LIN {X 0,Y 350.483,Z 210.53,A -85,B 0,C 180,E1 -14687.75,E2 -14687.75} C_VEL
LIN {X 0,Y 348.097,Z 207.912,A -85,B 0,C 180,E1 -14688.285,E2 -14688.285} C_VEL
LIN {X 0,Y 344.862,Z 203.942,A -85,B 0,C 180,E1 -14688.984,E2 -14688.984} C_VEL
LIN {X 0,Y 341.244,Z 199.767,A -85,B 0,C 180,E1 -14689.717,E2 -14689.717} C_VEL
LIN {X 0,Y 339.454,Z 197.486,A -85,B 0,C 180,E1 -14690.077,E2 -14690.077} C_VEL
LIN {X 0,Y 337.301,Z 194.627,A -85,B 0,C 180,E1 -14690.498,E2 -14690.498} C_VEL
LIN {X 0,Y 336.134,Z 192.909,A -85,B 0,C 180,E1 -14690.724,E2 -14690.724} C_VEL
LIN {X 0,Y 334.391,Z 190.698,A -85,B 0,C 180,E1 -14691.054,E2 -14691.054} C_VEL
LIN {X 0,Y 333.682,Z 188.419,A -85,B 0,C 180,E1 -14691.257,E2 -14691.257} C_VEL
LIN {X 0,Y 333.715,Z 188.414,A -85,B 0,C 180,E1 -14695.101,E2 -14695.101} C_VEL
LIN {X 0,Y 333.718,Z 188.416,A -85,B 0,C 180,E1 -14697.811,E2 -14697.811} C_VEL
LIN {X 0,Y 333.695,Z 188.419,A -85,B 0,C 180,E1 -14700.362,E2 -14700.362} C_VEL
LIN {X 0,Y 333.669,Z 188.42,A -85,B 0,C 180,E1 -14704.659,E2 -14704.659} C_VEL
LIN {X 0,Y 333.652,Z 188.425,A -85,B 0,C 180,E1 -14707.65,E2 -14707.65} C_VEL
LIN {X 0,Y 333.65,Z 188.421,A -85,B 0,C 180,E1 -14710.766,E2 -14710.766} C_VEL
LIN {X 0,Y 333.598,Z 188.429,A -85,B 0,C 180,E1 -14714.252,E2 -14714.252} C_VEL
LIN {X 0,Y 333.663,Z 188.425,A -85,B 0,C 180,E1 -14717.623,E2 -14717.623} C_VEL
LIN {X 0,Y 333.672,Z 188.422,A -85,B 0,C 180,E1 -14721.197,E2 -14721.197} C_VEL
LIN {X 0,Y 333.68,Z 188.422,A -85,B 0,C 180,E1 -14725.226,E2 -14725.226} C_VEL
LIN {X 0,Y 333.692,Z 188.418,A -85,B 0,C 180,E1 -14729.638,E2 -14729.638} C_VEL
LIN {X 0,Y 333.739,Z 188.411,A -85,B 0,C 180,E1 -14732.402,E2 -14732.402} C_VEL
LIN {X 0,Y 333.721,Z 188.417,A -85,B 0,C 180,E1 -14735.091,E2 -14735.091} C_VEL
LIN {X 0,Y 333.68,Z 188.421,A -85,B 0,C 180,E1 -14739.02,E2 -14739.02} C_VEL
LIN {X 0,Y 333.699,Z 188.414,A -85,B 0,C 180,E1 -14739.925,E2 -14739.925} C_VEL
LIN {X 0,Y 333.087,Z 188.496,A -85,B 0,C 180,E1 -14740.932,E2 -14740.932} C_VEL
LIN {X 0,Y 330.262,Z 188.848,A -85,B 0,C 180,E1 -14742.571,E2 -14742.571} C_VEL
LIN {X 0,Y 327.848,Z 189.149,A -85,B 0,C 180,E1 -14743.899,E2 -14743.899} C_VEL
LIN {X 0,Y 326.826,Z 189.275,A -85,B 0,C 180,E1 -14744.927,E2 -14744.927} C_VEL
LIN {X 0,Y 326.752,Z 189.281,A -85,B 0,C 180,E1 -14745.275,E2 -14745.275} C_VEL
LIN {X 0,Y 326.764,Z 189.282,A -85,B 0,C 180,E1 -14748.839,E2 -14748.839} C_VEL
LIN {X 0,Y 326.953,Z 189.261,A -85,B 0,C 180,E1 -14752.59,E2 -14752.59} C_VEL
LIN {X 0,Y 326.77,Z 189.277,A -85,B 0,C 180,E1 -14755.065,E2 -14755.065} C_VEL
LIN {X 0,Y 327.041,Z 189.24,A -85,B 0,C 180,E1 -14757.537,E2 -14757.537} C_VEL
LIN {X 0,Y 327.193,Z 189.225,A -85,B 0,C 180,E1 -14760.001,E2 -14760.001} C_VEL
LIN {X 0,Y 327.04,Z 189.248,A -85,B 0,C 180,E1 -14762.464,E2 -14762.464} C_VEL
LIN {X 0,Y 326.984,Z 189.257,A -85,B 0,C 180,E1 -14766.17,E2 -14766.17} C_VEL
LIN {X 0,Y 326.802,Z 189.279,A -85,B 0,C 180,E1 -14769.907,E2 -14769.907} C_VEL
LIN {X 0,Y 326.755,Z 189.284,A -85,B 0,C 180,E1 -14773.686,E2 -14773.686} C_VEL
LIN {X 0,Y 326.696,Z 189.291,A -85,B 0,C 180,E1 -14777.529,E2 -14777.529} C_VEL
LIN {X 0,Y 326.659,Z 189.294,A -85,B 0,C 180,E1 -14780.136,E2 -14780.136} C_VEL
LIN {X 0,Y 326.65,Z 189.295,A -85,B 0,C 180,E1 -14784.13,E2 -14784.13} C_VEL
LIN {X 0,Y 326.68,Z 189.291,A -85,B 0,C 180,E1 -14786.859,E2 -14786.859} C_VEL
LIN {X 0,Y 326.632,Z 189.297,A -85,B 0,C 180,E1 -14790.61,E2 -14790.61} C_VEL
LIN {X 0,Y 326.605,Z 189.302,A -85,B 0,C 180,E1 -14794.02,E2 -14794.02} C_VEL
LIN {X 0,Y 326.685,Z 189.697,A -85,B 0,C 180,E1 -14795.511,E2 -14795.511} C_VEL
LIN {X 0,Y 327.059,Z 192.418,A -85,B 0,C 180,E1 -14799.324,E2 -14799.324} C_VEL
LIN {X 0,Y 327.355,Z 194.259,A -85,B 0,C 180,E1 -14801.725,E2 -14801.725} C_VEL
LIN {X 0,Y 327.712,Z 196.982,A -85,B 0,C 180,E1 -14805.049,E2 -14805.049} C_VEL
LIN {X 0,Y 327.836,Z 199.974,A -85,B 0,C 180,E1 -14808.352,E2 -14808.352} C_VEL
LIN {X 0,Y 327.498,Z 203.094,A -85,B 0,C 180,E1 -14811.514,E2 -14811.514} C_VEL
LIN {X 0,Y 327.023,Z 206.495,A -85,B 0,C 180,E1 -14814.752,E2 -14814.752} C_VEL
LIN {X 0,Y 326.604,Z 209.457,A -85,B 0,C 180,E1 -14817.456,E2 -14817.456} C_VEL
LIN {X 0,Y 326.202,Z 212.67,A -85,B 0,C 180,E1 -14820.296,E2 -14820.296} C_VEL
LIN {X 0,Y 325.859,Z 215.915,A -85,B 0,C 180,E1 -14823.069,E2 -14823.069} C_VEL
LIN {X 0,Y 325.459,Z 220.798,A -85,B 0,C 180,E1 -14827.127,E2 -14827.127} C_VEL
LIN {X 0,Y 325.414,Z 221.412,A -85,B 0,C 180,E1 -14827.655,E2 -14827.655} C_VEL
LIN {X 0,Y 327.617,Z 230.715,A -85,B 0,C 180,E1 -14828.173,E2 -14828.173} C_VEL
LIN {X 0,Y 329.57,Z 240.233,A -85,B 0,C 180,E1 -14828.813,E2 -14828.813} C_VEL
LIN {X 0,Y 331.05,Z 249.851,A -85,B 0,C 180,E1 -14829.573,E2 -14829.573} C_VEL
LIN {X 0,Y 332.04,Z 258.46,A -85,B 0,C 180,E1 -14830.366,E2 -14830.366} C_VEL
LIN {X 0,Y 332.381,Z 263.384,A -85,B 0,C 180,E1 -14830.869,E2 -14830.869} C_VEL
LIN {X 0,Y 330.862,Z 275.575,A -85,B 0,C 180,E1 -14832.221,E2 -14832.221} C_VEL
LIN {X 0,Y 329.888,Z 283.327,A -85,B 0,C 180,E1 -14833.286,E2 -14833.286} C_VEL
LIN {X 0,Y 328.677,Z 292.466,A -85,B 0,C 180,E1 -14834.815,E2 -14834.815} C_VEL
LIN {X 0,Y 327.865,Z 298.672,A -85,B 0,C 180,E1 -14836.046,E2 -14836.046} C_VEL
LIN {X 0,Y 326.878,Z 305.21,A -85,B 0,C 180,E1 -14837.584,E2 -14837.584} C_VEL
LIN {X 0,Y 326.347,Z 309.716,A -85,B 0,C 180,E1 -14838.824,E2 -14838.824} C_VEL
LIN {X 0,Y 325.644,Z 315.21,A -85,B 0,C 180,E1 -14840.685,E2 -14840.685} C_VEL
LIN {X 0,Y 325.21,Z 319.539,A -85,B 0,C 180,E1 -14842.55,E2 -14842.55} C_VEL
LIN {X 0,Y 324.998,Z 322.39,A -85,B 0,C 180,E1 -14844.125,E2 -14844.125} C_VEL
LIN {X 0,Y 324.912,Z 325.1,A -85,B 0,C 180,E1 -14846.279,E2 -14846.279} C_VEL
LIN {X 0,Y 324.838,Z 326.158,A -85,B 0,C 180,E1 -14847.52,E2 -14847.52} C_VEL
LIN {X 0,Y 324.815,Z 326.747,A -85,B 0,C 180,E1 -14848.76,E2 -14848.76} C_VEL
LIN {X 0,Y 324.815,Z 326.747,A -85,B 0,C 180,E1 -14851.24,E2 -14851.24} C_VEL
LIN {X 0,Y 324.838,Z 326.158,A -85,B 0,C 180,E1 -14852.48,E2 -14852.48} C_VEL
LIN {X 0,Y 324.931,Z 323.709,A -85,B 0,C 180,E1 -14854.963,E2 -14854.963} C_VEL
LIN {X 0,Y 325.121,Z 320.757,A -85,B 0,C 180,E1 -14856.828,E2 -14856.828} C_VEL
LIN {X 0,Y 325.474,Z 316.766,A -85,B 0,C 180,E1 -14858.694,E2 -14858.694} C_VEL
LIN {X 0,Y 326.08,Z 311.633,A -85,B 0,C 180,E1 -14860.556,E2 -14860.556} C_VEL
LIN {X 0,Y 326.724,Z 306.367,A -85,B 0,C 180,E1 -14862.106,E2 -14862.106} C_VEL
LIN {X 0,Y 327.646,Z 300.048,A -85,B 0,C 180,E1 -14863.647,E2 -14863.647} C_VEL
LIN {X 0,Y 328.437,Z 294.094,A -85,B 0,C 180,E1 -14864.879,E2 -14864.879} C_VEL
LIN {X 0,Y 329.422,Z 287.165,A -85,B 0,C 180,E1 -14866.102,E2 -14866.102} C_VEL
LIN {X 0,Y 330.396,Z 278.98,A -85,B 0,C 180,E1 -14867.325,E2 -14867.325} C_VEL
LIN {X 0,Y 331.502,Z 270.468,A -85,B 0,C 180,E1 -14868.382,E2 -14868.382} C_VEL
LIN {X 0,Y 332.359,Z 263.383,A -85,B 0,C 180,E1 -14869.133,E2 -14869.133} C_VEL
LIN {X 0,Y 331.643,Z 254.402,A -85,B 0,C 180,E1 -14870.026,E2 -14870.026} C_VEL
LIN {X 0,Y 330.252,Z 244.324,A -85,B 0,C 180,E1 -14870.884,E2 -14870.884} C_VEL
LIN {X 0,Y 328.126,Z 233.062,A -85,B 0,C 180,E1 -14871.682,E2 -14871.682} C_VEL
LIN {X 0,Y 325.67,Z 223.147,A -85,B 0,C 180,E1 -14872.27,E2 -14872.27} C_VEL
LIN {X 0,Y 325.411,Z 221.414,A -85,B 0,C 180,E1 -14872.344,E2 -14872.344} C_VEL
LIN {X 0,Y 325.716,Z 217.555,A -85,B 0,C 180,E1 -14875.565,E2 -14875.565} C_VEL
LIN {X 0,Y 326.057,Z 214.284,A -85,B 0,C 180,E1 -14878.307,E2 -14878.307} C_VEL
LIN {X 0,Y 326.604,Z 209.433,A -85,B 0,C 180,E1 -14882.544,E2 -14882.544} C_VEL
LIN {X 0,Y 327.05,Z 206.248,A -85,B 0,C 180,E1 -14885.464,E2 -14885.464} C_VEL
LIN {X 0,Y 327.497,Z 203.094,A -85,B 0,C 180,E1 -14888.486,E2 -14888.486} C_VEL
LIN {X 0,Y 327.829,Z 199.972,A -85,B 0,C 180,E1 -14891.649,E2 -14891.649} C_VEL
LIN {X 0,Y 327.833,Z 198.426,A -85,B 0,C 180,E1 -14893.314,E2 -14893.314} C_VEL
LIN {X 0,Y 327.512,Z 195.562,A -85,B 0,C 180,E1 -14896.631,E2 -14896.631} C_VEL
LIN {X 0,Y 327.137,Z 193.006,A -85,B 0,C 180,E1 -14899.871,E2 -14899.871} C_VEL
LIN {X 0,Y 326.805,Z 190.726,A -85,B 0,C 180,E1 -14902.976,E2 -14902.976} C_VEL
LIN {X 0,Y 326.67,Z 189.471,A -85,B 0,C 180,E1 -14904.837,E2 -14904.837} C_VEL
LIN {X 0,Y 326.606,Z 189.302,A -85,B 0,C 180,E1 -14907.455,E2 -14907.455} C_VEL
LIN {X 0,Y 326.646,Z 189.298,A -85,B 0,C 180,E1 -14910.339,E2 -14910.339} C_VEL
LIN {X 0,Y 326.688,Z 189.295,A -85,B 0,C 180,E1 -14914.515,E2 -14914.515} C_VEL
LIN {X 0,Y 326.643,Z 189.299,A -85,B 0,C 180,E1 -14918.544,E2 -14918.544} C_VEL
LIN {X 0,Y 326.742,Z 189.282,A -85,B 0,C 180,E1 -14921.177,E2 -14921.177} C_VEL
LIN {X 0,Y 326.76,Z 189.28,A -85,B 0,C 180,E1 -14925.432,E2 -14925.432} C_VEL
LIN {X 0,Y 326.766,Z 189.279,A -85,B 0,C 180,E1 -14928.838,E2 -14928.838} C_VEL
LIN {X 0,Y 326.953,Z 189.256,A -85,B 0,C 180,E1 -14932.589,E2 -14932.589} C_VEL
LIN {X 0,Y 326.769,Z 189.279,A -85,B 0,C 180,E1 -14935.064,E2 -14935.064} C_VEL
LIN {X 0,Y 327.04,Z 189.248,A -85,B 0,C 180,E1 -14937.536,E2 -14937.536} C_VEL
LIN {X 0,Y 327.193,Z 189.225,A -85,B 0,C 180,E1 -14939.999,E2 -14939.999} C_VEL
LIN {X 0,Y 327.041,Z 189.24,A -85,B 0,C 180,E1 -14942.463,E2 -14942.463} C_VEL
LIN {X 0,Y 326.954,Z 189.255,A -85,B 0,C 180,E1 -14946.646,E2 -14946.646} C_VEL
LIN {X 0,Y 326.8,Z 189.275,A -85,B 0,C 180,E1 -14949.906,E2 -14949.906} C_VEL
LIN {X 0,Y 326.754,Z 189.281,A -85,B 0,C 180,E1 -14953.685,E2 -14953.685} C_VEL
LIN {X 0,Y 326.694,Z 189.29,A -85,B 0,C 180,E1 -14957.527,E2 -14957.527} C_VEL
LIN {X 0,Y 326.66,Z 189.29,A -85,B 0,C 180,E1 -14960.134,E2 -14960.134} C_VEL
LIN {X 0,Y 326.646,Z 189.293,A -85,B 0,C 180,E1 -14964.128,E2 -14964.128} C_VEL
LIN {X 0,Y 326.68,Z 189.294,A -85,B 0,C 180,E1 -14966.857,E2 -14966.857} C_VEL
LIN {X 0,Y 326.633,Z 189.299,A -85,B 0,C 180,E1 -14970.611,E2 -14970.611} C_VEL
LIN {X 0,Y 326.601,Z 189.3,A -85,B 0,C 180,E1 -14974.019,E2 -14974.019} C_VEL
LIN {X 0,Y 326.624,Z 189.297,A -85,B 0,C 180,E1 -14977.239,E2 -14977.239} C_VEL
LIN {X 0,Y 326.598,Z 189.303,A -85,B 0,C 180,E1 -14980.207,E2 -14980.207} C_VEL
LIN {X 0,Y 326.566,Z 189.304,A -85,B 0,C 180,E1 -14983.524,E2 -14983.524} C_VEL
LIN {X 0,Y 326.571,Z 189.303,A -85,B 0,C 180,E1 -14987.028,E2 -14987.028} C_VEL
LIN {X 0,Y 326.606,Z 189.3,A -85,B 0,C 180,E1 -14990.773,E2 -14990.773} C_VEL
LIN {X 0,Y 326.608,Z 189.301,A -85,B 0,C 180,E1 -14994.48,E2 -14994.48} C_VEL
LIN {X 0,Y 326.61,Z 189.3,A -85,B 0,C 180,E1 -14997.456,E2 -14997.456} C_VEL
LIN {X 0,Y 326.657,Z 189.295,A -85,B 0,C 180,E1 -15000.341,E2 -15000.341} C_VEL
LIN {X 0,Y 326.681,Z 189.291,A -85,B 0,C 180,E1 -15003.143,E2 -15003.143} C_VEL
LIN {X 0,Y 326.648,Z 189.299,A -85,B 0,C 180,E1 -15005.871,E2 -15005.871} C_VEL
LIN {X 0,Y 326.654,Z 189.298,A -85,B 0,C 180,E1 -15007.82,E2 -15007.82} C_VEL
LIN {X 0,Y 327.795,Z 192.347,A -85,B 0,C 180,E1 -15008.061,E2 -15008.061} C_VEL
LIN {X 0,Y 329.517,Z 194.65,A -85,B 0,C 180,E1 -15008.362,E2 -15008.362} C_VEL
LIN {X 0,Y 331.953,Z 198.098,A -85,B 0,C 180,E1 -15008.797,E2 -15008.797} C_VEL
LIN {X 0,Y 335.943,Z 203.215,A -85,B 0,C 180,E1 -15009.532,E2 -15009.532} C_VEL
LIN {X 0,Y 340.414,Z 208.614,A -85,B 0,C 180,E1 -15010.402,E2 -15010.402} C_VEL
LIN {X 0,Y 345.28,Z 214.213,A -85,B 0,C 180,E1 -15011.406,E2 -15011.406} C_VEL
LIN {X 0,Y 347.897,Z 217.095,A -85,B 0,C 180,E1 -15011.984,E2 -15011.984} C_VEL
LIN {X 0,Y 352.051,Z 221.223,A -85,B 0,C 180,E1 -15012.932,E2 -15012.932} C_VEL
LIN {X 0,Y 356.881,Z 226.359,A -85,B 0,C 180,E1 -15014.144,E2 -15014.144} C_VEL
LIN {X 0,Y 360.132,Z 229.27,A -85,B 0,C 180,E1 -15015.015,E2 -15015.015} C_VEL
LIN {X 0,Y 364.662,Z 233.73,A -85,B 0,C 180,E1 -15016.357,E2 -15016.357} C_VEL
LIN {X 0,Y 367.666,Z 236.169,A -85,B 0,C 180,E1 -15017.32,E2 -15017.32} C_VEL
LIN {X 0,Y 370.754,Z 239.393,A -85,B 0,C 180,E1 -15018.471,E2 -15018.471} C_VEL
LIN {X 0,Y 372.501,Z 240.811,A -85,B 0,C 180,E1 -15019.125,E2 -15019.125} C_VEL
LIN {X 0,Y 375.48,Z 242.667,A -85,B 0,C 180,E1 -15020.302,E2 -15020.302} C_VEL
LIN {X 0,Y 377.708,Z 245.024,A -85,B 0,C 180,E1 -15021.44,E2 -15021.44} C_VEL
LIN {X 0,Y 379.626,Z 247.006,A -85,B 0,C 180,E1 -15022.554,E2 -15022.554} C_VEL
LIN {X 0,Y 381.687,Z 248.584,A -85,B 0,C 180,E1 -15023.874,E2 -15023.874} C_VEL
LIN {X 0,Y 382.853,Z 249.33,A -85,B 0,C 180,E1 -15024.734,E2 -15024.734} C_VEL
LIN {X 0,Y 384.103,Z 249.928,A -85,B 0,C 180,E1 -15025.803,E2 -15025.803} C_VEL
LIN {X 0,Y 385.142,Z 250.169,A -85,B 0,C 180,E1 -15026.862,E2 -15026.862} C_VEL
LIN {X 0,Y 385.884,Z 250.348,A -85,B 0,C 180,E1 -15027.913,E2 -15027.913} C_VEL
LIN {X 0,Y 386.362,Z 250.4,A -85,B 0,C 180,E1 -15028.958,E2 -15028.958} C_VEL
LIN {X 0,Y 386.509,Z 250.455,A -85,B 0,C 180,E1 -15030,E2 -15030} C_VEL
LIN {X 0,Y 386.362,Z 250.371,A -85,B 0,C 180,E1 -15031.042,E2 -15031.042} C_VEL
LIN {X 0,Y 385.884,Z 250.332,A -85,B 0,C 180,E1 -15032.087,E2 -15032.087} C_VEL
LIN {X 0,Y 385.152,Z 250.141,A -85,B 0,C 180,E1 -15033.138,E2 -15033.138} C_VEL
LIN {X 0,Y 384.128,Z 249.9,A -85,B 0,C 180,E1 -15034.197,E2 -15034.197} C_VEL
LIN {X 0,Y 382.819,Z 249.345,A -85,B 0,C 180,E1 -15035.267,E2 -15035.267} C_VEL
LIN {X 0,Y 381.358,Z 248.36,A -85,B 0,C 180,E1 -15036.348,E2 -15036.348} C_VEL
LIN {X 0,Y 379.625,Z 246.957,A -85,B 0,C 180,E1 -15037.446,E2 -15037.446} C_VEL
LIN {X 0,Y 377.041,Z 244.248,A -85,B 0,C 180,E1 -15038.922,E2 -15038.922} C_VEL
LIN {X 0,Y 375.403,Z 242.649,A -85,B 0,C 180,E1 -15039.7,E2 -15039.7} C_VEL
LIN {X 0,Y 372.239,Z 240.59,A -85,B 0,C 180,E1 -15040.959,E2 -15040.959} C_VEL
LIN {X 0,Y 368.635,Z 237.327,A -85,B 0,C 180,E1 -15042.312,E2 -15042.312} C_VEL
LIN {X 0,Y 366.406,Z 235.019,A -85,B 0,C 180,E1 -15043.098,E2 -15043.098} C_VEL
LIN {X 0,Y 362.568,Z 231.873,A -85,B 0,C 180,E1 -15044.261,E2 -15044.261} C_VEL
LIN {X 0,Y 358.361,Z 227.539,A -85,B 0,C 180,E1 -15045.468,E2 -15045.468} C_VEL
LIN {X 0,Y 354.273,Z 223.764,A -85,B 0,C 180,E1 -15046.513,E2 -15046.513} C_VEL
LIN {X 0,Y 351.124,Z 220.432,A -85,B 0,C 180,E1 -15047.28,E2 -15047.28} C_VEL
LIN {X 0,Y 346.949,Z 215.921,A -85,B 0,C 180,E1 -15048.238,E2 -15048.238} C_VEL
LIN {X 0,Y 342.082,Z 210.601,A -85,B 0,C 180,E1 -15049.26,E2 -15049.26} C_VEL
LIN {X 0,Y 339.011,Z 207.141,A -85,B 0,C 180,E1 -15049.871,E2 -15049.871} C_VEL
LIN {X 0,Y 335.427,Z 202.682,A -85,B 0,C 180,E1 -15050.562,E2 -15050.562} C_VEL
LIN {X 0,Y 332.765,Z 198.959,A -85,B 0,C 180,E1 -15051.067,E2 -15051.067} C_VEL
LIN {X 0,Y 329.9,Z 195.384,A -85,B 0,C 180,E1 -15051.562,E2 -15051.562} C_VEL
LIN {X 0,Y 328.729,Z 193.458,A -85,B 0,C 180,E1 -15051.78,E2 -15051.78} C_VEL
LIN {X 0,Y 327.241,Z 191.338,A -85,B 0,C 180,E1 -15052.037,E2 -15052.037} C_VEL
LIN {X 0,Y 326.661,Z 189.297,A -85,B 0,C 180,E1 -15052.205,E2 -15052.205} C_VEL
LIN {X 0,Y 326.686,Z 189.29,A -85,B 0,C 180,E1 -15055.484,E2 -15055.484} C_VEL
LIN {X 0,Y 326.668,Z 189.296,A -85,B 0,C 180,E1 -15058.249,E2 -15058.249} C_VEL
LIN {X 0,Y 326.596,Z 189.3,A -85,B 0,C 180,E1 -15061.094,E2 -15061.094} C_VEL
LIN {X 0,Y 326.604,Z 189.304,A -85,B 0,C 180,E1 -15064.019,E2 -15064.019} C_VEL
LIN {X 0,Y 326.626,Z 189.297,A -85,B 0,C 180,E1 -15067.239,E2 -15067.239} C_VEL
LIN {X 0,Y 326.599,Z 189.302,A -85,B 0,C 180,E1 -15070.207,E2 -15070.207} C_VEL
LIN {X 0,Y 326.573,Z 189.306,A -85,B 0,C 180,E1 -15073.523,E2 -15073.523} C_VEL
LIN {X 0,Y 326.589,Z 189.302,A -85,B 0,C 180,E1 -15077.025,E2 -15077.025} C_VEL
LIN {X 0,Y 326.629,Z 189.296,A -85,B 0,C 180,E1 -15080.768,E2 -15080.768} C_VEL
LIN {X 0,Y 326.607,Z 189.299,A -85,B 0,C 180,E1 -15084.481,E2 -15084.481} C_VEL
LIN {X 0,Y 326.602,Z 189.303,A -85,B 0,C 180,E1 -15087.456,E2 -15087.456} C_VEL
LIN {X 0,Y 326.655,Z 189.293,A -85,B 0,C 180,E1 -15090.341,E2 -15090.341} C_VEL
LIN {X 0,Y 326.685,Z 189.289,A -85,B 0,C 180,E1 -15094.517,E2 -15094.517} C_VEL
LIN {X 0,Y 326.643,Z 189.296,A -85,B 0,C 180,E1 -15098.546,E2 -15098.546} C_VEL
LIN {X 0,Y 326.739,Z 189.285,A -85,B 0,C 180,E1 -15101.178,E2 -15101.178} C_VEL
LIN {X 0,Y 326.752,Z 189.281,A -85,B 0,C 180,E1 -15105.275,E2 -15105.275} C_VEL
LIN {X 0,Y 326.102,Z 189.364,A -85,B 0,C 180,E1 -15106.304,E2 -15106.304} C_VEL
LIN {X 0,Y 323.235,Z 189.719,A -85,B 0,C 180,E1 -15107.978,E2 -15107.978} C_VEL
LIN {X 0,Y 320.826,Z 190.018,A -85,B 0,C 180,E1 -15109.335,E2 -15109.335} C_VEL
LIN {X 0,Y 319.841,Z 190.144,A -85,B 0,C 180,E1 -15110.386,E2 -15110.386} C_VEL
LIN {X 0,Y 319.788,Z 190.146,A -85,B 0,C 180,E1 -15110.741,E2 -15110.741} C_VEL
LIN {X 0,Y 319.939,Z 190.129,A -85,B 0,C 180,E1 -15113.695,E2 -15113.695} C_VEL
LIN {X 0,Y 319.985,Z 190.117,A -85,B 0,C 180,E1 -15117.483,E2 -15117.483} C_VEL
LIN {X 0,Y 320.145,Z 190.102,A -85,B 0,C 180,E1 -15120.001,E2 -15120.001} C_VEL
LIN {X 0,Y 319.984,Z 190.127,A -85,B 0,C 180,E1 -15122.518,E2 -15122.518} C_VEL
LIN {X 0,Y 319.938,Z 190.133,A -85,B 0,C 180,E1 -15126.306,E2 -15126.306} C_VEL
LIN {X 0,Y 319.833,Z 190.143,A -85,B 0,C 180,E1 -15128.849,E2 -15128.849} C_VEL
LIN {X 0,Y 319.678,Z 190.162,A -85,B 0,C 180,E1 -15132.701,E2 -15132.701} C_VEL
LIN {X 0,Y 319.696,Z 190.161,A -85,B 0,C 180,E1 -15135.296,E2 -15135.296} C_VEL
LIN {X 0,Y 319.671,Z 190.164,A -85,B 0,C 180,E1 -15139.256,E2 -15139.256} C_VEL
LIN {X 0,Y 319.568,Z 190.179,A -85,B 0,C 180,E1 -15143.32,E2 -15143.32} C_VEL
LIN {X 0,Y 319.632,Z 190.169,A -85,B 0,C 180,E1 -15146.089,E2 -15146.089} C_VEL
LIN {X 0,Y 319.578,Z 190.177,A -85,B 0,C 180,E1 -15148.935,E2 -15148.935} C_VEL
LIN {X 0,Y 319.529,Z 190.185,A -85,B 0,C 180,E1 -15151.863,E2 -15151.863} C_VEL
LIN {X 0,Y 319.627,Z 190.434,A -85,B 0,C 180,E1 -15154.869,E2 -15154.869} C_VEL
LIN {X 0,Y 319.929,Z 192.541,A -85,B 0,C 180,E1 -15157.959,E2 -15157.959} C_VEL
LIN {X 0,Y 320.345,Z 195.316,A -85,B 0,C 180,E1 -15161.763,E2 -15161.763} C_VEL
LIN {X 0,Y 320.687,Z 198.349,A -85,B 0,C 180,E1 -15165.47,E2 -15165.47} C_VEL
LIN {X 0,Y 320.811,Z 200.725,A -85,B 0,C 180,E1 -15168.146,E2 -15168.146} C_VEL
LIN {X 0,Y 320.592,Z 202.992,A -85,B 0,C 180,E1 -15170.526,E2 -15170.526} C_VEL
LIN {X 0,Y 320.009,Z 206.864,A -85,B 0,C 180,E1 -15174.351,E2 -15174.351} C_VEL
LIN {X 0,Y 319.408,Z 210.912,A -85,B 0,C 180,E1 -15178.125,E2 -15178.125} C_VEL
LIN {X 0,Y 318.97,Z 215.028,A -85,B 0,C 180,E1 -15181.805,E2 -15181.805} C_VEL
LIN {X 0,Y 318.553,Z 218.987,A -85,B 0,C 180,E1 -15185.217,E2 -15185.217} C_VEL
LIN {X 0,Y 318.391,Z 221.196,A -85,B 0,C 180,E1 -15187.115,E2 -15187.115} C_VEL
LIN {X 0,Y 321.765,Z 235.746,A -85,B 0,C 180,E1 -15188.007,E2 -15188.007} C_VEL
LIN {X 0,Y 324.009,Z 248.649,A -85,B 0,C 180,E1 -15189.029,E2 -15189.029} C_VEL
LIN {X 0,Y 325.107,Z 258.24,A -85,B 0,C 180,E1 -15189.93,E2 -15189.93} C_VEL
LIN {X 0,Y 325.496,Z 264.783,A -85,B 0,C 180,E1 -15190.612,E2 -15190.612} C_VEL
LIN {X 0,Y 324.082,Z 275.363,A -85,B 0,C 180,E1 -15191.837,E2 -15191.837} C_VEL
LIN {X 0,Y 323.017,Z 283.496,A -85,B 0,C 180,E1 -15192.984,E2 -15192.984} C_VEL
LIN {X 0,Y 322.049,Z 290.806,A -85,B 0,C 180,E1 -15194.206,E2 -15194.206} C_VEL
LIN {X 0,Y 320.965,Z 298.461,A -85,B 0,C 180,E1 -15195.739,E2 -15195.739} C_VEL
LIN {X 0,Y 319.921,Z 304.998,A -85,B 0,C 180,E1 -15197.31,E2 -15197.31} C_VEL
LIN {X 0,Y 319.328,Z 309.503,A -85,B 0,C 180,E1 -15198.576,E2 -15198.576} C_VEL
LIN {X 0,Y 318.624,Z 314.999,A -85,B 0,C 180,E1 -15200.478,E2 -15200.478} C_VEL
LIN {X 0,Y 318.145,Z 319.327,A -85,B 0,C 180,E1 -15202.384,E2 -15202.384} C_VEL
LIN {X 0,Y 317.889,Z 322.474,A -85,B 0,C 180,E1 -15204.203,E2 -15204.203} C_VEL
LIN {X 0,Y 317.821,Z 324.888,A -85,B 0,C 180,E1 -15206.196,E2 -15206.196} C_VEL
LIN {X 0,Y 317.76,Z 325.947,A -85,B 0,C 180,E1 -15207.465,E2 -15207.465} C_VEL
LIN {X 0,Y 317.728,Z 326.536,A -85,B 0,C 180,E1 -15208.733,E2 -15208.733} C_VEL
LIN {X 0,Y 317.728,Z 326.536,A -85,B 0,C 180,E1 -15211.267,E2 -15211.267} C_VEL
LIN {X 0,Y 317.76,Z 325.947,A -85,B 0,C 180,E1 -15212.535,E2 -15212.535} C_VEL
LIN {X 0,Y 317.847,Z 323.498,A -85,B 0,C 180,E1 -15215.074,E2 -15215.074} C_VEL
LIN {X 0,Y 318.064,Z 320.546,A -85,B 0,C 180,E1 -15216.98,E2 -15216.98} C_VEL
LIN {X 0,Y 318.425,Z 316.553,A -85,B 0,C 180,E1 -15218.888,E2 -15218.888} C_VEL
LIN {X 0,Y 319.066,Z 311.42,A -85,B 0,C 180,E1 -15220.791,E2 -15220.791} C_VEL
LIN {X 0,Y 319.762,Z 306.155,A -85,B 0,C 180,E1 -15222.374,E2 -15222.374} C_VEL
LIN {X 0,Y 320.739,Z 299.837,A -85,B 0,C 180,E1 -15223.947,E2 -15223.947} C_VEL
LIN {X 0,Y 321.551,Z 293.881,A -85,B 0,C 180,E1 -15225.205,E2 -15225.205} C_VEL
LIN {X 0,Y 322.534,Z 286.952,A -85,B 0,C 180,E1 -15226.455,E2 -15226.455} C_VEL
LIN {X 0,Y 323.598,Z 278.768,A -85,B 0,C 180,E1 -15227.701,E2 -15227.701} C_VEL
LIN {X 0,Y 324.771,Z 270.257,A -85,B 0,C 180,E1 -15228.777,E2 -15228.777} C_VEL
LIN {X 0,Y 325.553,Z 263.168,A -85,B 0,C 180,E1 -15229.549,E2 -15229.549} C_VEL
LIN {X 0,Y 324.509,Z 252.66,A -85,B 0,C 180,E1 -15230.61,E2 -15230.61} C_VEL
LIN {X 0,Y 323.105,Z 243.169,A -85,B 0,C 180,E1 -15231.429,E2 -15231.429} C_VEL
LIN {X 0,Y 321.092,Z 232.659,A -85,B 0,C 180,E1 -15232.19,E2 -15232.19} C_VEL
LIN {X 0,Y 318.358,Z 221.21,A -85,B 0,C 180,E1 -15232.875,E2 -15232.875} C_VEL
LIN {X 0,Y 318.673,Z 217.356,A -85,B 0,C 180,E1 -15236.172,E2 -15236.172} C_VEL
LIN {X 0,Y 319.034,Z 214.113,A -85,B 0,C 180,E1 -15238.988,E2 -15238.988} C_VEL
LIN {X 0,Y 319.408,Z 210.9,A -85,B 0,C 180,E1 -15241.875,E2 -15241.875} C_VEL
LIN {X 0,Y 320.007,Z 206.861,A -85,B 0,C 180,E1 -15245.649,E2 -15245.649} C_VEL
LIN {X 0,Y 320.593,Z 202.991,A -85,B 0,C 180,E1 -15249.474,E2 -15249.474} C_VEL
LIN {X 0,Y 320.803,Z 199.883,A -85,B 0,C 180,E1 -15252.775,E2 -15252.775} C_VEL
LIN {X 0,Y 320.509,Z 196.817,A -85,B 0,C 180,E1 -15256.353,E2 -15256.353} C_VEL
LIN {X 0,Y 320.284,Z 194.873,A -85,B 0,C 180,E1 -15258.83,E2 -15258.83} C_VEL
LIN {X 0,Y 319.854,Z 192.357,A -85,B 0,C 180,E1 -15262.279,E2 -15262.279} C_VEL
LIN {X 0,Y 319.637,Z 190.421,A -85,B 0,C 180,E1 -15265.132,E2 -15265.132} C_VEL
LIN {X 0,Y 319.529,Z 190.184,A -85,B 0,C 180,E1 -15268.137,E2 -15268.137} C_VEL
LIN {X 0,Y 319.609,Z 190.172,A -85,B 0,C 180,E1 -15271.589,E2 -15271.589} C_VEL
LIN {X 0,Y 319.602,Z 190.173,A -85,B 0,C 180,E1 -15275.303,E2 -15275.303} C_VEL
LIN {X 0,Y 319.594,Z 190.177,A -85,B 0,C 180,E1 -15278.047,E2 -15278.047} C_VEL
LIN {X 0,Y 319.686,Z 190.162,A -85,B 0,C 180,E1 -15280.962,E2 -15280.962} C_VEL
LIN {X 0,Y 319.728,Z 190.156,A -85,B 0,C 180,E1 -15285.275,E2 -15285.275} C_VEL
LIN {X 0,Y 319.749,Z 190.158,A -85,B 0,C 180,E1 -15289.872,E2 -15289.872} C_VEL
LIN {X 0,Y 319.908,Z 190.134,A -85,B 0,C 180,E1 -15292.425,E2 -15292.425} C_VEL
LIN {X 0,Y 319.739,Z 190.154,A -85,B 0,C 180,E1 -15294.955,E2 -15294.955} C_VEL
LIN {X 0,Y 319.984,Z 190.127,A -85,B 0,C 180,E1 -15297.482,E2 -15297.482} C_VEL
LIN {X 0,Y 320.145,Z 190.102,A -85,B 0,C 180,E1 -15299.999,E2 -15299.999} C_VEL
LIN {X 0,Y 319.985,Z 190.117,A -85,B 0,C 180,E1 -15302.517,E2 -15302.517} C_VEL
LIN {X 0,Y 319.916,Z 190.131,A -85,B 0,C 180,E1 -15306.634,E2 -15306.634} C_VEL
LIN {X 0,Y 319.747,Z 190.152,A -85,B 0,C 180,E1 -15310.127,E2 -15310.127} C_VEL
LIN {X 0,Y 319.726,Z 190.156,A -85,B 0,C 180,E1 -15314.724,E2 -15314.724} C_VEL
LIN {X 0,Y 319.684,Z 190.166,A -85,B 0,C 180,E1 -15319.037,E2 -15319.037} C_VEL
LIN {X 0,Y 319.565,Z 190.178,A -85,B 0,C 180,E1 -15323.319,E2 -15323.319} C_VEL
LIN {X 0,Y 319.63,Z 190.167,A -85,B 0,C 180,E1 -15326.088,E2 -15326.088} C_VEL
LIN {X 0,Y 319.585,Z 190.178,A -85,B 0,C 180,E1 -15328.933,E2 -15328.933} C_VEL
LIN {X 0,Y 319.527,Z 190.181,A -85,B 0,C 180,E1 -15331.861,E2 -15331.861} C_VEL
LIN {X 0,Y 319.574,Z 190.175,A -85,B 0,C 180,E1 -15335.543,E2 -15335.543} C_VEL
LIN {X 0,Y 319.577,Z 190.176,A -85,B 0,C 180,E1 -15338.006,E2 -15338.006} C_VEL
LIN {X 0,Y 319.561,Z 190.177,A -85,B 0,C 180,E1 -15341.605,E2 -15341.605} C_VEL
LIN {X 0,Y 319.484,Z 190.186,A -85,B 0,C 180,E1 -15345.257,E2 -15345.257} C_VEL
LIN {X 0,Y 319.523,Z 190.183,A -85,B 0,C 180,E1 -15348.712,E2 -15348.712} C_VEL
LIN {X 0,Y 319.572,Z 190.179,A -85,B 0,C 180,E1 -15352.344,E2 -15352.344} C_VEL
LIN {X 0,Y 319.556,Z 190.177,A -85,B 0,C 180,E1 -15355.123,E2 -15355.123} C_VEL
LIN {X 0,Y 319.57,Z 190.176,A -85,B 0,C 180,E1 -15359.057,E2 -15359.057} C_VEL
LIN {X 0,Y 319.613,Z 190.171,A -85,B 0,C 180,E1 -15362.499,E2 -15362.499} C_VEL
LIN {X 0,Y 319.601,Z 190.174,A -85,B 0,C 180,E1 -15365.304,E2 -15365.304} C_VEL
LIN {X 0,Y 319.569,Z 190.178,A -85,B 0,C 180,E1 -15367.015,E2 -15367.015} C_VEL
LIN {X 0,Y 320.7,Z 193.22,A -85,B 0,C 180,E1 -15367.231,E2 -15367.231} C_VEL
LIN {X 0,Y 322.464,Z 195.872,A -85,B 0,C 180,E1 -15367.501,E2 -15367.501} C_VEL
LIN {X 0,Y 327.552,Z 203.078,A -85,B 0,C 180,E1 -15368.33,E2 -15368.33} C_VEL
LIN {X 0,Y 332.308,Z 208.966,A -85,B 0,C 180,E1 -15369.177,E2 -15369.177} C_VEL
LIN {X 0,Y 336.686,Z 214.216,A -85,B 0,C 180,E1 -15370.017,E2 -15370.017} C_VEL
LIN {X 0,Y 341.977,Z 220.215,A -85,B 0,C 180,E1 -15371.106,E2 -15371.106} C_VEL
LIN {X 0,Y 347.387,Z 226.079,A -85,B 0,C 180,E1 -15372.334,E2 -15372.334} C_VEL
LIN {X 0,Y 350.149,Z 228.859,A -85,B 0,C 180,E1 -15372.991,E2 -15372.991} C_VEL
LIN {X 0,Y 354.817,Z 233.478,A -85,B 0,C 180,E1 -15374.197,E2 -15374.197} C_VEL
LIN {X 0,Y 356.924,Z 235.405,A -85,B 0,C 180,E1 -15374.757,E2 -15374.757} C_VEL
LIN {X 0,Y 360.433,Z 239.028,A -85,B 0,C 180,E1 -15375.813,E2 -15375.813} C_VEL
LIN {X 0,Y 364.942,Z 242.843,A -85,B 0,C 180,E1 -15377.235,E2 -15377.235} C_VEL
LIN {X 0,Y 367.798,Z 245.743,A -85,B 0,C 180,E1 -15378.304,E2 -15378.304} C_VEL
LIN {X 0,Y 371.446,Z 248.362,A -85,B 0,C 180,E1 -15379.692,E2 -15379.692} C_VEL
LIN {X 0,Y 373.743,Z 250.205,A -85,B 0,C 180,E1 -15380.711,E2 -15380.711} C_VEL
LIN {X 0,Y 376.856,Z 253.511,A -85,B 0,C 180,E1 -15382.499,E2 -15382.499} C_VEL
LIN {X 0,Y 378.589,Z 254.913,A -85,B 0,C 180,E1 -15383.605,E2 -15383.605} C_VEL
LIN {X 0,Y 380.813,Z 256.207,A -85,B 0,C 180,E1 -15385.254,E2 -15385.254} C_VEL
LIN {X 0,Y 382.489,Z 256.731,A -85,B 0,C 180,E1 -15386.84,E2 -15386.84} C_VEL
LIN {X 0,Y 383.25,Z 256.938,A -85,B 0,C 180,E1 -15387.898,E2 -15387.898} C_VEL
LIN {X 0,Y 383.748,Z 256.978,A -85,B 0,C 180,E1 -15388.951,E2 -15388.951} C_VEL
LIN {X 0,Y 383.89,Z 257.041,A -85,B 0,C 180,E1 -15390,E2 -15390} C_VEL
LIN {X 0,Y 383.74,Z 256.968,A -85,B 0,C 180,E1 -15391.049,E2 -15391.049} C_VEL
LIN {X 0,Y 383.246,Z 256.925,A -85,B 0,C 180,E1 -15392.102,E2 -15392.102} C_VEL
LIN {X 0,Y 382.496,Z 256.712,A -85,B 0,C 180,E1 -15393.16,E2 -15393.16} C_VEL
LIN {X 0,Y 380.814,Z 256.19,A -85,B 0,C 180,E1 -15394.748,E2 -15394.748} C_VEL
LIN {X 0,Y 378.599,Z 254.874,A -85,B 0,C 180,E1 -15396.395,E2 -15396.395} C_VEL
LIN {X 0,Y 376.111,Z 252.73,A -85,B 0,C 180,E1 -15397.969,E2 -15397.969} C_VEL
LIN {X 0,Y 372.703,Z 249.234,A -85,B 0,C 180,E1 -15399.771,E2 -15399.771} C_VEL
LIN {X 0,Y 369.741,Z 247.312,A -85,B 0,C 180,E1 -15400.957,E2 -15400.957} C_VEL
LIN {X 0,Y 366.522,Z 244.539,A -85,B 0,C 180,E1 -15402.176,E2 -15402.176} C_VEL
LIN {X 0,Y 361.785,Z 240.177,A -85,B 0,C 180,E1 -15403.764,E2 -15403.764} C_VEL
LIN {X 0,Y 356.926,Z 235.389,A -85,B 0,C 180,E1 -15405.244,E2 -15405.244} C_VEL
LIN {X 0,Y 351.032,Z 229.857,A -85,B 0,C 180,E1 -15406.779,E2 -15406.779} C_VEL
LIN {X 0,Y 347.835,Z 226.469,A -85,B 0,C 180,E1 -15407.566,E2 -15407.566} C_VEL
LIN {X 0,Y 343.368,Z 221.669,A -85,B 0,C 180,E1 -15408.592,E2 -15408.592} C_VEL
LIN {X 0,Y 338.444,Z 216.304,A -85,B 0,C 180,E1 -15409.624,E2 -15409.624} C_VEL
LIN {X 0,Y 333.053,Z 209.887,A -85,B 0,C 180,E1 -15410.684,E2 -15410.684} C_VEL
LIN {X 0,Y 328.834,Z 204.638,A -85,B 0,C 180,E1 -15411.451,E2 -15411.451} C_VEL
LIN {X 0,Y 325.101,Z 199.688,A -85,B 0,C 180,E1 -15412.08,E2 -15412.08} C_VEL
LIN {X 0,Y 322.039,Z 195.103,A -85,B 0,C 180,E1 -15412.571,E2 -15412.571} C_VEL
LIN {X 0,Y 319.973,Z 191.74,A -85,B 0,C 180,E1 -15412.882,E2 -15412.882} C_VEL
LIN {X 0,Y 319.578,Z 190.176,A -85,B 0,C 180,E1 -15413.003,E2 -15413.003} C_VEL
LIN {X 0,Y 319.631,Z 190.173,A -85,B 0,C 180,E1 -15416.088,E2 -15416.088} C_VEL
LIN {X 0,Y 319.594,Z 190.173,A -85,B 0,C 180,E1 -15418.933,E2 -15418.933} C_VEL
LIN {X 0,Y 319.534,Z 190.184,A -85,B 0,C 180,E1 -15421.861,E2 -15421.861} C_VEL
LIN {X 0,Y 319.576,Z 190.177,A -85,B 0,C 180,E1 -15425.543,E2 -15425.543} C_VEL
LIN {X 0,Y 319.594,Z 190.177,A -85,B 0,C 180,E1 -15428.004,E2 -15428.004} C_VEL
LIN {X 0,Y 319.563,Z 190.18,A -85,B 0,C 180,E1 -15431.606,E2 -15431.606} C_VEL
LIN {X 0,Y 319.488,Z 190.187,A -85,B 0,C 180,E1 -15435.258,E2 -15435.258} C_VEL
LIN {X 0,Y 319.537,Z 190.18,A -85,B 0,C 180,E1 -15438.714,E2 -15438.714} C_VEL
LIN {X 0,Y 319.576,Z 190.175,A -85,B 0,C 180,E1 -15442.343,E2 -15442.343} C_VEL
LIN {X 0,Y 319.555,Z 190.18,A -85,B 0,C 180,E1 -15445.124,E2 -15445.124} C_VEL
LIN {X 0,Y 319.565,Z 190.18,A -85,B 0,C 180,E1 -15449.058,E2 -15449.058} C_VEL
LIN {X 0,Y 319.603,Z 190.172,A -85,B 0,C 180,E1 -15452.499,E2 -15452.499} C_VEL
LIN {X 0,Y 319.6,Z 190.174,A -85,B 0,C 180,E1 -15455.304,E2 -15455.304} C_VEL
LIN {X 0,Y 319.592,Z 190.172,A -85,B 0,C 180,E1 -15458.048,E2 -15458.048} C_VEL
LIN {X 0,Y 319.684,Z 190.166,A -85,B 0,C 180,E1 -15460.963,E2 -15460.963} C_VEL
LIN {X 0,Y 319.726,Z 190.156,A -85,B 0,C 180,E1 -15465.276,E2 -15465.276} C_VEL
LIN {X 0,Y 319.747,Z 190.152,A -85,B 0,C 180,E1 -15469.873,E2 -15469.873} C_VEL
LIN {X 0,Y 319.788,Z 190.146,A -85,B 0,C 180,E1 -15470.741,E2 -15470.741} C_VEL
LIN {X 0,Y 319.511,Z 190.184,A -85,B 0,C 180,E1 -15471.445,E2 -15471.445} C_VEL
LIN {X 0,Y 317.54,Z 190.436,A -85,B 0,C 180,E1 -15472.823,E2 -15472.823} C_VEL
LIN {X 0,Y 313.739,Z 190.91,A -85,B 0,C 180,E1 -15474.888,E2 -15474.888} C_VEL
LIN {X 0,Y 312.751,Z 191.026,A -85,B 0,C 180,E1 -15475.964,E2 -15475.964} C_VEL
LIN {X 0,Y 312.713,Z 191.027,A -85,B 0,C 180,E1 -15476.328,E2 -15476.328} C_VEL
LIN {X 0,Y 312.985,Z 190.993,A -85,B 0,C 180,E1 -15478.714,E2 -15478.714} C_VEL
LIN {X 0,Y 312.985,Z 190.994,A -85,B 0,C 180,E1 -15481.287,E2 -15481.287} C_VEL
LIN {X 0,Y 312.71,Z 191.03,A -85,B 0,C 180,E1 -15485.158,E2 -15485.158} C_VEL
LIN {X 0,Y 312.849,Z 191.015,A -85,B 0,C 180,E1 -15487.747,E2 -15487.747} C_VEL
LIN {X 0,Y 312.665,Z 191.038,A -85,B 0,C 180,E1 -15491.672,E2 -15491.672} C_VEL
LIN {X 0,Y 312.697,Z 191.032,A -85,B 0,C 180,E1 -15494.888,E2 -15494.888} C_VEL
LIN {X 0,Y 312.627,Z 191.042,A -85,B 0,C 180,E1 -15499.237,E2 -15499.237} C_VEL
LIN {X 0,Y 312.543,Z 191.051,A -85,B 0,C 180,E1 -15502.79,E2 -15502.79} C_VEL
LIN {X 0,Y 312.6,Z 191.046,A -85,B 0,C 180,E1 -15505.936,E2 -15505.936} C_VEL
LIN {X 0,Y 312.536,Z 191.057,A -85,B 0,C 180,E1 -15509.652,E2 -15509.652} C_VEL
LIN {X 0,Y 312.528,Z 191.057,A -85,B 0,C 180,E1 -15513.692,E2 -15513.692} C_VEL
LIN {X 0,Y 312.701,Z 192.307,A -85,B 0,C 180,E1 -15515.993,E2 -15515.993} C_VEL
LIN {X 0,Y 312.984,Z 194.322,A -85,B 0,C 180,E1 -15518.958,E2 -15518.958} C_VEL
LIN {X 0,Y 313.383,Z 196.789,A -85,B 0,C 180,E1 -15522.283,E2 -15522.283} C_VEL
LIN {X 0,Y 313.686,Z 199.802,A -85,B 0,C 180,E1 -15526.01,E2 -15526.01} C_VEL
LIN {X 0,Y 313.76,Z 201.339,A -85,B 0,C 180,E1 -15527.781,E2 -15527.781} C_VEL
LIN {X 0,Y 313.437,Z 204.444,A -85,B 0,C 180,E1 -15531.111,E2 -15531.111} C_VEL
LIN {X 0,Y 312.982,Z 207.587,A -85,B 0,C 180,E1 -15534.28,E2 -15534.28} C_VEL
LIN {X 0,Y 312.461,Z 210.77,A -85,B 0,C 180,E1 -15537.329,E2 -15537.329} C_VEL
LIN {X 0,Y 311.911,Z 215.275,A -85,B 0,C 180,E1 -15541.493,E2 -15541.493} C_VEL
LIN {X 0,Y 311.536,Z 218.813,A -85,B 0,C 180,E1 -15544.62,E2 -15544.62} C_VEL
LIN {X 0,Y 311.344,Z 221.034,A -85,B 0,C 180,E1 -15546.592,E2 -15546.592} C_VEL
LIN {X 0,Y 313.673,Z 230.711,A -85,B 0,C 180,E1 -15547.171,E2 -15547.171} C_VEL
LIN {X 0,Y 315.578,Z 239.405,A -85,B 0,C 180,E1 -15547.799,E2 -15547.799} C_VEL
LIN {X 0,Y 317.293,Z 250.044,A -85,B 0,C 180,E1 -15548.699,E2 -15548.699} C_VEL
LIN {X 0,Y 318.331,Z 259.664,A -85,B 0,C 180,E1 -15549.652,E2 -15549.652} C_VEL
LIN {X 0,Y 318.733,Z 264.569,A -85,B 0,C 180,E1 -15550.183,E2 -15550.183} C_VEL
LIN {X 0,Y 317.305,Z 275.151,A -85,B 0,C 180,E1 -15551.435,E2 -15551.435} C_VEL
LIN {X 0,Y 316.255,Z 282.899,A -85,B 0,C 180,E1 -15552.542,E2 -15552.542} C_VEL
LIN {X 0,Y 315.146,Z 290.959,A -85,B 0,C 180,E1 -15553.925,E2 -15553.925} C_VEL
LIN {X 0,Y 314.058,Z 298.248,A -85,B 0,C 180,E1 -15555.419,E2 -15555.419} C_VEL
LIN {X 0,Y 312.981,Z 304.786,A -85,B 0,C 180,E1 -15557.024,E2 -15557.024} C_VEL
LIN {X 0,Y 312.323,Z 309.29,A -85,B 0,C 180,E1 -15558.316,E2 -15558.316} C_VEL
LIN {X 0,Y 311.586,Z 314.786,A -85,B 0,C 180,E1 -15560.261,E2 -15560.261} C_VEL
LIN {X 0,Y 311.071,Z 319.114,A -85,B 0,C 180,E1 -15562.209,E2 -15562.209} C_VEL
LIN {X 0,Y 310.899,Z 321.485,A -85,B 0,C 180,E1 -15563.51,E2 -15563.51} C_VEL
LIN {X 0,Y 310.765,Z 323.286,A -85,B 0,C 180,E1 -15564.81,E2 -15564.81} C_VEL
LIN {X 0,Y 310.684,Z 325.736,A -85,B 0,C 180,E1 -15567.407,E2 -15567.407} C_VEL
LIN {X 0,Y 310.643,Z 326.325,A -85,B 0,C 180,E1 -15568.704,E2 -15568.704} C_VEL
LIN {X 0,Y 310.643,Z 326.325,A -85,B 0,C 180,E1 -15571.296,E2 -15571.296} C_VEL
LIN {X 0,Y 310.684,Z 325.736,A -85,B 0,C 180,E1 -15572.593,E2 -15572.593} C_VEL
LIN {X 0,Y 310.767,Z 323.286,A -85,B 0,C 180,E1 -15575.19,E2 -15575.19} C_VEL
LIN {X 0,Y 311.001,Z 320.334,A -85,B 0,C 180,E1 -15577.14,E2 -15577.14} C_VEL
LIN {X 0,Y 311.397,Z 316.341,A -85,B 0,C 180,E1 -15579.09,E2 -15579.09} C_VEL
LIN {X 0,Y 312.06,Z 311.208,A -85,B 0,C 180,E1 -15581.036,E2 -15581.036} C_VEL
LIN {X 0,Y 312.78,Z 305.942,A -85,B 0,C 180,E1 -15582.655,E2 -15582.655} C_VEL
LIN {X 0,Y 313.825,Z 299.625,A -85,B 0,C 180,E1 -15584.261,E2 -15584.261} C_VEL
LIN {X 0,Y 314.687,Z 293.67,A -85,B 0,C 180,E1 -15585.545,E2 -15585.545} C_VEL
LIN {X 0,Y 315.676,Z 286.739,A -85,B 0,C 180,E1 -15586.823,E2 -15586.823} C_VEL
LIN {X 0,Y 316.816,Z 278.556,A -85,B 0,C 180,E1 -15588.093,E2 -15588.093} C_VEL
LIN {X 0,Y 318.044,Z 270.045,A -85,B 0,C 180,E1 -15589.19,E2 -15589.19} C_VEL
LIN {X 0,Y 318.743,Z 264.569,A -85,B 0,C 180,E1 -15589.816,E2 -15589.816} C_VEL
LIN {X 0,Y 317.735,Z 253.508,A -85,B 0,C 180,E1 -15590.98,E2 -15590.98} C_VEL
LIN {X 0,Y 316.152,Z 242.649,A -85,B 0,C 180,E1 -15591.944,E2 -15591.944} C_VEL
LIN {X 0,Y 314.067,Z 232.235,A -85,B 0,C 180,E1 -15592.724,E2 -15592.724} C_VEL
LIN {X 0,Y 311.378,Z 221.738,A -85,B 0,C 180,E1 -15593.382,E2 -15593.382} C_VEL
LIN {X 0,Y 311.311,Z 221.006,A -85,B 0,C 180,E1 -15593.431,E2 -15593.431} C_VEL
LIN {X 0,Y 311.661,Z 217.157,A -85,B 0,C 180,E1 -15596.808,E2 -15596.808} C_VEL
LIN {X 0,Y 312.048,Z 213.942,A -85,B 0,C 180,E1 -15599.701,E2 -15599.701} C_VEL
LIN {X 0,Y 312.628,Z 209.653,A -85,B 0,C 180,E1 -15603.718,E2 -15603.718} C_VEL
LIN {X 0,Y 313.183,Z 206.007,A -85,B 0,C 180,E1 -15607.293,E2 -15607.293} C_VEL
LIN {X 0,Y 313.651,Z 202.884,A -85,B 0,C 180,E1 -15610.526,E2 -15610.526} C_VEL
LIN {X 0,Y 313.757,Z 201.229,A -85,B 0,C 180,E1 -15612.337,E2 -15612.337} C_VEL
LIN {X 0,Y 313.528,Z 198.248,A -85,B 0,C 180,E1 -15615.832,E2 -15615.832} C_VEL
LIN {X 0,Y 313.164,Z 195.493,A -85,B 0,C 180,E1 -15619.396,E2 -15619.396} C_VEL
LIN {X 0,Y 312.796,Z 193.232,A -85,B 0,C 180,E1 -15622.652,E2 -15622.652} C_VEL
LIN {X 0,Y 312.543,Z 191.16,A -85,B 0,C 180,E1 -15625.794,E2 -15625.794} C_VEL
LIN {X 0,Y 312.518,Z 191.058,A -85,B 0,C 180,E1 -15628.853,E2 -15628.853} C_VEL
LIN {X 0,Y 312.568,Z 191.049,A -85,B 0,C 180,E1 -15631.823,E2 -15631.823} C_VEL
LIN {X 0,Y 312.583,Z 191.051,A -85,B 0,C 180,E1 -15634.71,E2 -15634.71} C_VEL
LIN {X 0,Y 312.585,Z 191.048,A -85,B 0,C 180,E1 -15637.528,E2 -15637.528} C_VEL
LIN {X 0,Y 312.635,Z 191.041,A -85,B 0,C 180,E1 -15641.656,E2 -15641.656} C_VEL
LIN {X 0,Y 312.69,Z 191.034,A -85,B 0,C 180,E1 -15645.685,E2 -15645.685} C_VEL
LIN {X 0,Y 312.695,Z 191.034,A -85,B 0,C 180,E1 -15649.641,E2 -15649.641} C_VEL
LIN {X 0,Y 312.849,Z 191.015,A -85,B 0,C 180,E1 -15652.253,E2 -15652.253} C_VEL
LIN {X 0,Y 312.709,Z 191.03,A -85,B 0,C 180,E1 -15654.842,E2 -15654.842} C_VEL
LIN {X 0,Y 312.985,Z 190.994,A -85,B 0,C 180,E1 -15658.713,E2 -15658.713} C_VEL
LIN {X 0,Y 312.985,Z 190.993,A -85,B 0,C 180,E1 -15661.286,E2 -15661.286} C_VEL
LIN {X 0,Y 312.71,Z 191.03,A -85,B 0,C 180,E1 -15665.157,E2 -15665.157} C_VEL
LIN {X 0,Y 312.848,Z 191.015,A -85,B 0,C 180,E1 -15667.746,E2 -15667.746} C_VEL
LIN {X 0,Y 312.664,Z 191.038,A -85,B 0,C 180,E1 -15671.671,E2 -15671.671} C_VEL
LIN {X 0,Y 312.695,Z 191.033,A -85,B 0,C 180,E1 -15674.887,E2 -15674.887} C_VEL
LIN {X 0,Y 312.625,Z 191.042,A -85,B 0,C 180,E1 -15679.236,E2 -15679.236} C_VEL
LIN {X 0,Y 312.541,Z 191.054,A -85,B 0,C 180,E1 -15682.789,E2 -15682.789} C_VEL
LIN {X 0,Y 312.578,Z 191.049,A -85,B 0,C 180,E1 -15686.722,E2 -15686.722} C_VEL
LIN {X 0,Y 312.54,Z 191.051,A -85,B 0,C 180,E1 -15689.65,E2 -15689.65} C_VEL
LIN {X 0,Y 312.514,Z 191.054,A -85,B 0,C 180,E1 -15693.689,E2 -15693.689} C_VEL
LIN {X 0,Y 312.535,Z 191.052,A -85,B 0,C 180,E1 -15697.383,E2 -15697.383} C_VEL
LIN {X 0,Y 312.494,Z 191.06,A -85,B 0,C 180,E1 -15700.707,E2 -15700.707} C_VEL
LIN {X 0,Y 312.45,Z 191.066,A -85,B 0,C 180,E1 -15704.209,E2 -15704.209} C_VEL
LIN {X 0,Y 312.479,Z 191.061,A -85,B 0,C 180,E1 -15707.919,E2 -15707.919} C_VEL
LIN {X 0,Y 312.53,Z 191.056,A -85,B 0,C 180,E1 -15711.91,E2 -15711.91} C_VEL
LIN {X 0,Y 312.502,Z 191.06,A -85,B 0,C 180,E1 -15715.79,E2 -15715.79} C_VEL
LIN {X 0,Y 312.524,Z 191.054,A -85,B 0,C 180,E1 -15718.854,E2 -15718.854} C_VEL
LIN {X 0,Y 312.58,Z 191.051,A -85,B 0,C 180,E1 -15721.826,E2 -15721.826} C_VEL
LIN {X 0,Y 312.581,Z 191.047,A -85,B 0,C 180,E1 -15724.711,E2 -15724.711} C_VEL
LIN {X 0,Y 312.526,Z 191.056,A -85,B 0,C 180,E1 -15726.328,E2 -15726.328} C_VEL
LIN {X 0,Y 313.592,Z 194.019,A -85,B 0,C 180,E1 -15726.526,E2 -15726.526} C_VEL
LIN {X 0,Y 316.624,Z 198.931,A -85,B 0,C 180,E1 -15726.948,E2 -15726.948} C_VEL
LIN {X 0,Y 319.716,Z 203.512,A -85,B 0,C 180,E1 -15727.403,E2 -15727.403} C_VEL
LIN {X 0,Y 323.571,Z 208.713,A -85,B 0,C 180,E1 -15728.035,E2 -15728.035} C_VEL
LIN {X 0,Y 328.149,Z 214.408,A -85,B 0,C 180,E1 -15728.843,E2 -15728.843} C_VEL
LIN {X 0,Y 332.786,Z 219.917,A -85,B 0,C 180,E1 -15729.729,E2 -15729.729} C_VEL
LIN {X 0,Y 338.079,Z 225.926,A -85,B 0,C 180,E1 -15730.833,E2 -15730.833} C_VEL
LIN {X 0,Y 343.893,Z 232.156,A -85,B 0,C 180,E1 -15732.149,E2 -15732.149} C_VEL
LIN {X 0,Y 349.934,Z 238.344,A -85,B 0,C 180,E1 -15733.67,E2 -15733.67} C_VEL
LIN {X 0,Y 352.582,Z 240.564,A -85,B 0,C 180,E1 -15734.348,E2 -15734.348} C_VEL
LIN {X 0,Y 356.981,Z 245.168,A -85,B 0,C 180,E1 -15735.673,E2 -15735.673} C_VEL
LIN {X 0,Y 361.497,Z 249.007,A -85,B 0,C 180,E1 -15737.111,E2 -15737.111} C_VEL
LIN {X 0,Y 365.587,Z 252.894,A -85,B 0,C 180,E1 -15738.639,E2 -15738.639} C_VEL
LIN {X 0,Y 369.445,Z 255.469,A -85,B 0,C 180,E1 -15740.142,E2 -15740.142} C_VEL
LIN {X 0,Y 371.647,Z 257.82,A -85,B 0,C 180,E1 -15741.299,E2 -15741.299} C_VEL
LIN {X 0,Y 373.543,Z 259.76,A -85,B 0,C 180,E1 -15742.432,E2 -15742.432} C_VEL
LIN {X 0,Y 375.299,Z 261.193,A -85,B 0,C 180,E1 -15743.549,E2 -15743.549} C_VEL
LIN {X 0,Y 376.832,Z 262.146,A -85,B 0,C 180,E1 -15744.649,E2 -15744.649} C_VEL
LIN {X 0,Y 378.138,Z 262.767,A -85,B 0,C 180,E1 -15745.737,E2 -15745.737} C_VEL
LIN {X 0,Y 379.841,Z 263.199,A -85,B 0,C 180,E1 -15747.599,E2 -15747.599} C_VEL
LIN {X 0,Y 380.536,Z 263.296,A -85,B 0,C 180,E1 -15748.942,E2 -15748.942} C_VEL
LIN {X 0,Y 380.672,Z 263.369,A -85,B 0,C 180,E1 -15750,E2 -15750} C_VEL
LIN {X 0,Y 380.525,Z 263.291,A -85,B 0,C 180,E1 -15751.058,E2 -15751.058} C_VEL
LIN {X 0,Y 379.839,Z 263.212,A -85,B 0,C 180,E1 -15752.394,E2 -15752.394} C_VEL
LIN {X 0,Y 378.155,Z 262.762,A -85,B 0,C 180,E1 -15754.263,E2 -15754.263} C_VEL
LIN {X 0,Y 376.837,Z 262.174,A -85,B 0,C 180,E1 -15755.351,E2 -15755.351} C_VEL
LIN {X 0,Y 375.009,Z 260.894,A -85,B 0,C 180,E1 -15756.659,E2 -15756.659} C_VEL
LIN {X 0,Y 373.57,Z 259.764,A -85,B 0,C 180,E1 -15757.567,E2 -15757.567} C_VEL
LIN {X 0,Y 370.399,Z 256.484,A -85,B 0,C 180,E1 -15759.375,E2 -15759.375} C_VEL
LIN {X 0,Y 368.083,Z 254.622,A -85,B 0,C 180,E1 -15760.384,E2 -15760.384} C_VEL
LIN {X 0,Y 365.579,Z 252.886,A -85,B 0,C 180,E1 -15761.355,E2 -15761.355} C_VEL
LIN {X 0,Y 363.127,Z 250.717,A -85,B 0,C 180,E1 -15762.292,E2 -15762.292} C_VEL
LIN {X 0,Y 359.519,Z 247.16,A -85,B 0,C 180,E1 -15763.567,E2 -15763.567} C_VEL
LIN {X 0,Y 355.017,Z 243.271,A -85,B 0,C 180,E1 -15764.913,E2 -15764.913} C_VEL
LIN {X 0,Y 351.024,Z 239.229,A -85,B 0,C 180,E1 -15766.051,E2 -15766.051} C_VEL
LIN {X 0,Y 346.526,Z 234.874,A -85,B 0,C 180,E1 -15767.205,E2 -15767.205} C_VEL
LIN {X 0,Y 340.043,Z 228.095,A -85,B 0,C 180,E1 -15768.733,E2 -15768.733} C_VEL
LIN {X 0,Y 334.12,Z 221.481,A -85,B 0,C 180,E1 -15770.001,E2 -15770.001} C_VEL
LIN {X 0,Y 328.782,Z 215.2,A -85,B 0,C 180,E1 -15771.036,E2 -15771.036} C_VEL
LIN {X 0,Y 324.332,Z 209.675,A -85,B 0,C 180,E1 -15771.836,E2 -15771.836} C_VEL
LIN {X 0,Y 320.438,Z 204.537,A -85,B 0,C 180,E1 -15772.481,E2 -15772.481} C_VEL
LIN {X 0,Y 317.065,Z 199.63,A -85,B 0,C 180,E1 -15772.989,E2 -15772.989} C_VEL
LIN {X 0,Y 314.617,Z 195.668,A -85,B 0,C 180,E1 -15773.341,E2 -15773.341} C_VEL
LIN {X 0,Y 312.737,Z 192.06,A -85,B 0,C 180,E1 -15773.6,E2 -15773.6} C_VEL
LIN {X 0,Y 312.534,Z 191.054,A -85,B 0,C 180,E1 -15773.667,E2 -15773.667} C_VEL
LIN {X 0,Y 312.582,Z 191.048,A -85,B 0,C 180,E1 -15776.722,E2 -15776.722} C_VEL
LIN {X 0,Y 312.545,Z 191.053,A -85,B 0,C 180,E1 -15779.649,E2 -15779.649} C_VEL
LIN {X 0,Y 312.515,Z 191.057,A -85,B 0,C 180,E1 -15783.689,E2 -15783.689} C_VEL
LIN {X 0,Y 312.548,Z 191.052,A -85,B 0,C 180,E1 -15787.381,E2 -15787.381} C_VEL
LIN {X 0,Y 312.496,Z 191.056,A -85,B 0,C 180,E1 -15790.707,E2 -15790.707} C_VEL
LIN {X 0,Y 312.46,Z 191.062,A -85,B 0,C 180,E1 -15794.207,E2 -15794.207} C_VEL
LIN {X 0,Y 312.519,Z 191.056,A -85,B 0,C 180,E1 -15797.91,E2 -15797.91} C_VEL
LIN {X 0,Y 312.538,Z 191.053,A -85,B 0,C 180,E1 -15801.909,E2 -15801.909} C_VEL
LIN {X 0,Y 312.501,Z 191.057,A -85,B 0,C 180,E1 -15805.79,E2 -15805.79} C_VEL
LIN {X 0,Y 312.518,Z 191.056,A -85,B 0,C 180,E1 -15808.854,E2 -15808.854} C_VEL
LIN {X 0,Y 312.569,Z 191.048,A -85,B 0,C 180,E1 -15811.825,E2 -15811.825} C_VEL
LIN {X 0,Y 312.58,Z 191.047,A -85,B 0,C 180,E1 -15814.711,E2 -15814.711} C_VEL
LIN {X 0,Y 312.582,Z 191.047,A -85,B 0,C 180,E1 -15817.529,E2 -15817.529} C_VEL
LIN {X 0,Y 312.633,Z 191.04,A -85,B 0,C 180,E1 -15821.657,E2 -15821.657} C_VEL
LIN {X 0,Y 312.689,Z 191.031,A -85,B 0,C 180,E1 -15825.687,E2 -15825.687} C_VEL
LIN {X 0,Y 312.693,Z 191.031,A -85,B 0,C 180,E1 -15829.642,E2 -15829.642} C_VEL
LIN {X 0,Y 312.848,Z 191.015,A -85,B 0,C 180,E1 -15832.254,E2 -15832.254} C_VEL
LIN {X 0,Y 312.71,Z 191.03,A -85,B 0,C 180,E1 -15834.843,E2 -15834.843} C_VEL
LIN {X 0,Y 312.713,Z 191.027,A -85,B 0,C 180,E1 -15836.328,E2 -15836.328} C_VEL
LIN {X 0,Y 312.184,Z 191.089,A -85,B 0,C 180,E1 -15837.406,E2 -15837.406} C_VEL
LIN {X 0,Y 309.452,Z 191.43,A -85,B 0,C 180,E1 -15839.164,E2 -15839.164} C_VEL
LIN {X 0,Y 307.048,Z 191.737,A -85,B 0,C 180,E1 -15840.59,E2 -15840.59} C_VEL
LIN {X 0,Y 305.988,Z 191.867,A -85,B 0,C 180,E1 -15841.692,E2 -15841.692} C_VEL
LIN {X 0,Y 305.891,Z 191.877,A -85,B 0,C 180,E1 -15842.065,E2 -15842.065} C_VEL
LIN {X 0,Y 305.837,Z 191.888,A -85,B 0,C 180,E1 -15846.598,E2 -15846.598} C_VEL
LIN {X 0,Y 305.7,Z 191.904,A -85,B 0,C 180,E1 -15849.262,E2 -15849.262} C_VEL
LIN {X 0,Y 305.585,Z 191.919,A -85,B 0,C 180,E1 -15853.297,E2 -15853.297} C_VEL
LIN {X 0,Y 305.591,Z 191.921,A -85,B 0,C 180,E1 -15856.021,E2 -15856.021} C_VEL
LIN {X 0,Y 305.574,Z 191.922,A -85,B 0,C 180,E1 -15859.446,E2 -15859.446} C_VEL
LIN {X 0,Y 305.488,Z 191.931,A -85,B 0,C 180,E1 -15863.042,E2 -15863.042} C_VEL
LIN {X 0,Y 305.529,Z 191.926,A -85,B 0,C 180,E1 -15866.222,E2 -15866.222} C_VEL
LIN {X 0,Y 305.486,Z 191.934,A -85,B 0,C 180,E1 -15869.048,E2 -15869.048} C_VEL
LIN {X 0,Y 305.472,Z 191.937,A -85,B 0,C 180,E1 -15873.517,E2 -15873.517} C_VEL
LIN {X 0,Y 305.756,Z 193.879,A -85,B 0,C 180,E1 -15876.701,E2 -15876.701} C_VEL
LIN {X 0,Y 306.177,Z 196.687,A -85,B 0,C 180,E1 -15880.758,E2 -15880.758} C_VEL
LIN {X 0,Y 306.528,Z 199.71,A -85,B 0,C 180,E1 -15884.704,E2 -15884.704} C_VEL
LIN {X 0,Y 306.693,Z 201.747,A -85,B 0,C 180,E1 -15887.164,E2 -15887.164} C_VEL
LIN {X 0,Y 306.508,Z 204.33,A -85,B 0,C 180,E1 -15890.058,E2 -15890.058} C_VEL
LIN {X 0,Y 306.013,Z 207.609,A -85,B 0,C 180,E1 -15893.498,E2 -15893.498} C_VEL
LIN {X 0,Y 305.525,Z 210.612,A -85,B 0,C 180,E1 -15896.491,E2 -15896.491} C_VEL
LIN {X 0,Y 305.062,Z 213.798,A -85,B 0,C 180,E1 -15899.547,E2 -15899.547} C_VEL
LIN {X 0,Y 304.666,Z 217.025,A -85,B 0,C 180,E1 -15902.526,E2 -15902.526} C_VEL
LIN {X 0,Y 304.295,Z 220.821,A -85,B 0,C 180,E1 -15906.006,E2 -15906.006} C_VEL
LIN {X 0,Y 307.146,Z 232.488,A -85,B 0,C 180,E1 -15906.759,E2 -15906.759} C_VEL
LIN {X 0,Y 309.307,Z 242.996,A -85,B 0,C 180,E1 -15907.583,E2 -15907.583} C_VEL
LIN {X 0,Y 310.934,Z 254.279,A -85,B 0,C 180,E1 -15908.623,E2 -15908.623} C_VEL
LIN {X 0,Y 311.881,Z 265.777,A -85,B 0,C 180,E1 -15909.901,E2 -15909.901} C_VEL
LIN {X 0,Y 310.383,Z 276.073,A -85,B 0,C 180,E1 -15911.176,E2 -15911.176} C_VEL
LIN {X 0,Y 309.175,Z 284.607,A -85,B 0,C 180,E1 -15912.471,E2 -15912.471} C_VEL
LIN {X 0,Y 308.049,Z 292.26,A -85,B 0,C 180,E1 -15913.861,E2 -15913.861} C_VEL
LIN {X 0,Y 306.907,Z 299.412,A -85,B 0,C 180,E1 -15915.411,E2 -15915.411} C_VEL
LIN {X 0,Y 305.828,Z 305.73,A -85,B 0,C 180,E1 -15917.053,E2 -15917.053} C_VEL
LIN {X 0,Y 305.065,Z 310.996,A -85,B 0,C 180,E1 -15918.708,E2 -15918.708} C_VEL
LIN {X 0,Y 304.347,Z 316.129,A -85,B 0,C 180,E1 -15920.698,E2 -15920.698} C_VEL
LIN {X 0,Y 303.876,Z 320.12,A -85,B 0,C 180,E1 -15922.692,E2 -15922.692} C_VEL
LIN {X 0,Y 303.688,Z 323.075,A -85,B 0,C 180,E1 -15924.689,E2 -15924.689} C_VEL
LIN {X 0,Y 303.61,Z 325.526,A -85,B 0,C 180,E1 -15927.347,E2 -15927.347} C_VEL
LIN {X 0,Y 303.561,Z 326.114,A -85,B 0,C 180,E1 -15928.673,E2 -15928.673} C_VEL
LIN {X 0,Y 303.561,Z 326.114,A -85,B 0,C 180,E1 -15931.327,E2 -15931.327} C_VEL
LIN {X 0,Y 303.61,Z 325.526,A -85,B 0,C 180,E1 -15932.653,E2 -15932.653} C_VEL
LIN {X 0,Y 303.688,Z 323.075,A -85,B 0,C 180,E1 -15935.311,E2 -15935.311} C_VEL
LIN {X 0,Y 303.934,Z 320.122,A -85,B 0,C 180,E1 -15937.306,E2 -15937.306} C_VEL
LIN {X 0,Y 304.347,Z 316.129,A -85,B 0,C 180,E1 -15939.302,E2 -15939.302} C_VEL
LIN {X 0,Y 305.065,Z 310.996,A -85,B 0,C 180,E1 -15941.292,E2 -15941.292} C_VEL
LIN {X 0,Y 305.827,Z 305.73,A -85,B 0,C 180,E1 -15942.947,E2 -15942.947} C_VEL
LIN {X 0,Y 306.913,Z 299.412,A -85,B 0,C 180,E1 -15944.589,E2 -15944.589} C_VEL
LIN {X 0,Y 308.064,Z 292.243,A -85,B 0,C 180,E1 -15946.142,E2 -15946.142} C_VEL
LIN {X 0,Y 309.167,Z 284.607,A -85,B 0,C 180,E1 -15947.529,E2 -15947.529} C_VEL
LIN {X 0,Y 310.38,Z 276.073,A -85,B 0,C 180,E1 -15948.824,E2 -15948.824} C_VEL
LIN {X 0,Y 311.889,Z 265.777,A -85,B 0,C 180,E1 -15950.098,E2 -15950.098} C_VEL
LIN {X 0,Y 310.808,Z 253.248,A -85,B 0,C 180,E1 -15951.474,E2 -15951.474} C_VEL
LIN {X 0,Y 309.324,Z 243.025,A -85,B 0,C 180,E1 -15952.414,E2 -15952.414} C_VEL
LIN {X 0,Y 307.084,Z 232.089,A -85,B 0,C 180,E1 -15953.267,E2 -15953.267} C_VEL
LIN {X 0,Y 304.334,Z 221.376,A -85,B 0,C 180,E1 -15953.962,E2 -15953.962} C_VEL
LIN {X 0,Y 304.271,Z 220.804,A -85,B 0,C 180,E1 -15954.012,E2 -15954.012} C_VEL
LIN {X 0,Y 304.661,Z 216.978,A -85,B 0,C 180,E1 -15957.475,E2 -15957.475} C_VEL
LIN {X 0,Y 305.228,Z 212.607,A -85,B 0,C 180,E1 -15961.575,E2 -15961.575} C_VEL
LIN {X 0,Y 305.777,Z 209.022,A -85,B 0,C 180,E1 -15965.071,E2 -15965.071} C_VEL
LIN {X 0,Y 306.355,Z 205.447,A -85,B 0,C 180,E1 -15968.74,E2 -15968.74} C_VEL
LIN {X 0,Y 306.667,Z 202.775,A -85,B 0,C 180,E1 -15971.651,E2 -15971.651} C_VEL
LIN {X 0,Y 306.576,Z 200.168,A -85,B 0,C 180,E1 -15974.711,E2 -15974.711} C_VEL
LIN {X 0,Y 306.251,Z 197.383,A -85,B 0,C 180,E1 -15978.278,E2 -15978.278} C_VEL
LIN {X 0,Y 305.871,Z 194.977,A -85,B 0,C 180,E1 -15981.655,E2 -15981.655} C_VEL
LIN {X 0,Y 305.596,Z 192.868,A -85,B 0,C 180,E1 -15984.904,E2 -15984.904} C_VEL
LIN {X 0,Y 305.473,Z 191.937,A -85,B 0,C 180,E1 -15986.483,E2 -15986.483} C_VEL
LIN {X 0,Y 305.511,Z 191.929,A -85,B 0,C 180,E1 -15991.112,E2 -15991.112} C_VEL
LIN {X 0,Y 305.563,Z 191.924,A -85,B 0,C 180,E1 -15994.086,E2 -15994.086} C_VEL
LIN {X 0,Y 305.523,Z 191.931,A -85,B 0,C 180,E1 -15998.404,E2 -15998.404} C_VEL
LIN {X 0,Y 305.587,Z 191.918,A -85,B 0,C 180,E1 -16001.217,E2 -16001.217} C_VEL
LIN {X 0,Y 305.646,Z 191.91,A -85,B 0,C 180,E1 -16005.348,E2 -16005.348} C_VEL
LIN {X 0,Y 305.632,Z 191.913,A -85,B 0,C 180,E1 -16009.399,E2 -16009.399} C_VEL
LIN {X 0,Y 305.793,Z 191.895,A -85,B 0,C 180,E1 -16012.073,E2 -16012.073} C_VEL
LIN {X 0,Y 305.681,Z 191.906,A -85,B 0,C 180,E1 -16014.723,E2 -16014.723} C_VEL
LIN {X 0,Y 305.952,Z 191.87,A -85,B 0,C 180,E1 -16018.683,E2 -16018.683} C_VEL
LIN {X 0,Y 305.952,Z 191.868,A -85,B 0,C 180,E1 -16021.316,E2 -16021.316} C_VEL
LIN {X 0,Y 305.838,Z 191.886,A -85,B 0,C 180,E1 -16026.597,E2 -16026.597} C_VEL
LIN {X 0,Y 305.699,Z 191.906,A -85,B 0,C 180,E1 -16029.26,E2 -16029.26} C_VEL
LIN {X 0,Y 305.584,Z 191.922,A -85,B 0,C 180,E1 -16033.295,E2 -16033.295} C_VEL
LIN {X 0,Y 305.589,Z 191.917,A -85,B 0,C 180,E1 -16036.02,E2 -16036.02} C_VEL
LIN {X 0,Y 305.572,Z 191.919,A -85,B 0,C 180,E1 -16039.444,E2 -16039.444} C_VEL
LIN {X 0,Y 305.486,Z 191.934,A -85,B 0,C 180,E1 -16043.041,E2 -16043.041} C_VEL
LIN {X 0,Y 305.549,Z 191.922,A -85,B 0,C 180,E1 -16046.229,E2 -16046.229} C_VEL
LIN {X 0,Y 305.491,Z 191.933,A -85,B 0,C 180,E1 -16049.05,E2 -16049.05} C_VEL
LIN {X 0,Y 305.459,Z 191.933,A -85,B 0,C 180,E1 -16053.517,E2 -16053.517} C_VEL
LIN {X 0,Y 305.492,Z 191.933,A -85,B 0,C 180,E1 -16056.736,E2 -16056.736} C_VEL
LIN {X 0,Y 305.457,Z 191.938,A -85,B 0,C 180,E1 -16060.601,E2 -16060.601} C_VEL
LIN {X 0,Y 305.429,Z 191.937,A -85,B 0,C 180,E1 -16063.653,E2 -16063.653} C_VEL
LIN {X 0,Y 305.45,Z 191.934,A -85,B 0,C 180,E1 -16067.414,E2 -16067.414} C_VEL
LIN {X 0,Y 305.49,Z 191.931,A -85,B 0,C 180,E1 -16071.6,E2 -16071.6} C_VEL
LIN {X 0,Y 305.458,Z 191.934,A -85,B 0,C 180,E1 -16074.887,E2 -16074.887} C_VEL
LIN {X 0,Y 305.452,Z 191.937,A -85,B 0,C 180,E1 -16078.354,E2 -16078.354} C_VEL
LIN {X 0,Y 305.525,Z 191.926,A -85,B 0,C 180,E1 -16081.115,E2 -16081.115} C_VEL
LIN {X 0,Y 305.568,Z 191.924,A -85,B 0,C 180,E1 -16084.088,E2 -16084.088} C_VEL
LIN {X 0,Y 305.497,Z 191.933,A -85,B 0,C 180,E1 -16085.749,E2 -16085.749} C_VEL
LIN {X 0,Y 306.701,Z 195.1,A -85,B 0,C 180,E1 -16085.945,E2 -16085.945} C_VEL
LIN {X 0,Y 310.726,Z 202.438,A -85,B 0,C 180,E1 -16086.482,E2 -16086.482} C_VEL
LIN {X 0,Y 316.679,Z 211.087,A -85,B 0,C 180,E1 -16087.379,E2 -16087.379} C_VEL
LIN {X 0,Y 323.361,Z 219.332,A -85,B 0,C 180,E1 -16088.516,E2 -16088.516} C_VEL
LIN {X 0,Y 329.646,Z 226.769,A -85,B 0,C 180,E1 -16089.728,E2 -16089.728} C_VEL
LIN {X 0,Y 335.371,Z 233.093,A -85,B 0,C 180,E1 -16090.947,E2 -16090.947} C_VEL
LIN {X 0,Y 340.801,Z 238.805,A -85,B 0,C 180,E1 -16092.202,E2 -16092.202} C_VEL
LIN {X 0,Y 345.709,Z 243.9,A -85,B 0,C 180,E1 -16093.465,E2 -16093.465} C_VEL
LIN {X 0,Y 349.889,Z 247.839,A -85,B 0,C 180,E1 -16094.608,E2 -16094.608} C_VEL
LIN {X 0,Y 352.827,Z 250.834,A -85,B 0,C 180,E1 -16095.501,E2 -16095.501} C_VEL
LIN {X 0,Y 357.265,Z 254.577,A -85,B 0,C 180,E1 -16096.898,E2 -16096.898} C_VEL
LIN {X 0,Y 361.484,Z 258.606,A -85,B 0,C 180,E1 -16098.464,E2 -16098.464} C_VEL
LIN {X 0,Y 365.565,Z 261.392,A -85,B 0,C 180,E1 -16100.036,E2 -16100.036} C_VEL
LIN {X 0,Y 369.072,Z 265.049,A -85,B 0,C 180,E1 -16101.968,E2 -16101.968} C_VEL
LIN {X 0,Y 371.448,Z 267.112,A -85,B 0,C 180,E1 -16103.482,E2 -16103.482} C_VEL
LIN {X 0,Y 373.783,Z 268.512,A -85,B 0,C 180,E1 -16105.214,E2 -16105.214} C_VEL
LIN {X 0,Y 375.455,Z 269.071,A -85,B 0,C 180,E1 -16106.781,E2 -16106.781} C_VEL
LIN {X 0,Y 376.272,Z 269.294,A -85,B 0,C 180,E1 -16107.859,E2 -16107.859} C_VEL
LIN {X 0,Y 376.815,Z 269.352,A -85,B 0,C 180,E1 -16108.931,E2 -16108.931} C_VEL
LIN {X 0,Y 376.973,Z 269.399,A -85,B 0,C 180,E1 -16110,E2 -16110} C_VEL
LIN {X 0,Y 376.809,Z 269.339,A -85,B 0,C 180,E1 -16111.069,E2 -16111.069} C_VEL
LIN {X 0,Y 376.271,Z 269.27,A -85,B 0,C 180,E1 -16112.141,E2 -16112.141} C_VEL
LIN {X 0,Y 375.45,Z 269.057,A -85,B 0,C 180,E1 -16113.219,E2 -16113.219} C_VEL
LIN {X 0,Y 373.779,Z 268.504,A -85,B 0,C 180,E1 -16114.78,E2 -16114.78} C_VEL
LIN {X 0,Y 371.462,Z 267.059,A -85,B 0,C 180,E1 -16116.518,E2 -16116.518} C_VEL
LIN {X 0,Y 369.075,Z 265.041,A -85,B 0,C 180,E1 -16118.035,E2 -16118.035} C_VEL
LIN {X 0,Y 365.533,Z 261.441,A -85,B 0,C 180,E1 -16119.964,E2 -16119.964} C_VEL
LIN {X 0,Y 361.462,Z 258.6,A -85,B 0,C 180,E1 -16121.537,E2 -16121.537} C_VEL
LIN {X 0,Y 357.385,Z 254.751,A -85,B 0,C 180,E1 -16123.048,E2 -16123.048} C_VEL
LIN {X 0,Y 354.783,Z 252.449,A -85,B 0,C 180,E1 -16123.918,E2 -16123.918} C_VEL
LIN {X 0,Y 349.892,Z 247.828,A -85,B 0,C 180,E1 -16125.394,E2 -16125.394} C_VEL
LIN {X 0,Y 343.436,Z 241.64,A -85,B 0,C 180,E1 -16127.134,E2 -16127.134} C_VEL
LIN {X 0,Y 336.793,Z 234.786,A -85,B 0,C 180,E1 -16128.724,E2 -16128.724} C_VEL
LIN {X 0,Y 329.645,Z 226.77,A -85,B 0,C 180,E1 -16130.271,E2 -16130.271} C_VEL
LIN {X 0,Y 323.928,Z 220.007,A -85,B 0,C 180,E1 -16131.376,E2 -16131.376} C_VEL
LIN {X 0,Y 319.479,Z 214.5,A -85,B 0,C 180,E1 -16132.171,E2 -16132.171} C_VEL
LIN {X 0,Y 315.304,Z 208.994,A -85,B 0,C 180,E1 -16132.851,E2 -16132.851} C_VEL
LIN {X 0,Y 311.697,Z 203.735,A -85,B 0,C 180,E1 -16133.388,E2 -16133.388} C_VEL
LIN {X 0,Y 309.035,Z 199.504,A -85,B 0,C 180,E1 -16133.747,E2 -16133.747} C_VEL
LIN {X 0,Y 305.79,Z 193.272,A -85,B 0,C 180,E1 -16134.178,E2 -16134.178} C_VEL
LIN {X 0,Y 305.491,Z 191.934,A -85,B 0,C 180,E1 -16134.268,E2 -16134.268} C_VEL
LIN {X 0,Y 305.536,Z 191.925,A -85,B 0,C 180,E1 -16137.389,E2 -16137.389} C_VEL
LIN {X 0,Y 305.464,Z 191.936,A -85,B 0,C 180,E1 -16140.408,E2 -16140.408} C_VEL
LIN {X 0,Y 305.46,Z 191.938,A -85,B 0,C 180,E1 -16144.079,E2 -16144.079} C_VEL
LIN {X 0,Y 305.498,Z 191.929,A -85,B 0,C 180,E1 -16146.736,E2 -16146.736} C_VEL
LIN {X 0,Y 305.461,Z 191.935,A -85,B 0,C 180,E1 -16150.106,E2 -16150.106} C_VEL
LIN {X 0,Y 305.44,Z 191.94,A -85,B 0,C 180,E1 -16153.652,E2 -16153.652} C_VEL
LIN {X 0,Y 305.468,Z 191.933,A -85,B 0,C 180,E1 -16158.149,E2 -16158.149} C_VEL
LIN {X 0,Y 305.503,Z 191.932,A -85,B 0,C 180,E1 -16161.603,E2 -16161.603} C_VEL
LIN {X 0,Y 305.457,Z 191.935,A -85,B 0,C 180,E1 -16164.887,E2 -16164.887} C_VEL
LIN {X 0,Y 305.446,Z 191.935,A -85,B 0,C 180,E1 -16168.355,E2 -16168.355} C_VEL
LIN {X 0,Y 305.516,Z 191.931,A -85,B 0,C 180,E1 -16171.114,E2 -16171.114} C_VEL
LIN {X 0,Y 305.567,Z 191.919,A -85,B 0,C 180,E1 -16174.088,E2 -16174.088} C_VEL
LIN {X 0,Y 305.496,Z 191.93,A -85,B 0,C 180,E1 -16178.403,E2 -16178.403} C_VEL
LIN {X 0,Y 305.585,Z 191.92,A -85,B 0,C 180,E1 -16181.218,E2 -16181.218} C_VEL
LIN {X 0,Y 305.644,Z 191.91,A -85,B 0,C 180,E1 -16185.35,E2 -16185.35} C_VEL
LIN {X 0,Y 305.63,Z 191.911,A -85,B 0,C 180,E1 -16189.4,E2 -16189.4} C_VEL
LIN {X 0,Y 305.792,Z 191.893,A -85,B 0,C 180,E1 -16192.075,E2 -16192.075} C_VEL
LIN {X 0,Y 305.681,Z 191.906,A -85,B 0,C 180,E1 -16194.724,E2 -16194.724} C_VEL
LIN {X 0,Y 305.952,Z 191.868,A -85,B 0,C 180,E1 -16198.684,E2 -16198.684} C_VEL
LIN {X 0,Y 305.952,Z 191.87,A -85,B 0,C 180,E1 -16201.317,E2 -16201.317} C_VEL
LIN {X 0,Y 305.891,Z 191.877,A -85,B 0,C 180,E1 -16202.065,E2 -16202.065} C_VEL
LIN {X 0,Y 305.184,Z 191.969,A -85,B 0,C 180,E1 -16203.163,E2 -16203.163} C_VEL
LIN {X 0,Y 302.281,Z 192.329,A -85,B 0,C 180,E1 -16204.948,E2 -16204.948} C_VEL
LIN {X 0,Y 299.845,Z 192.636,A -85,B 0,C 180,E1 -16206.396,E2 -16206.396} C_VEL
LIN {X 0,Y 298.812,Z 192.762,A -85,B 0,C 180,E1 -16207.518,E2 -16207.518} C_VEL
LIN {X 0,Y 298.733,Z 192.774,A -85,B 0,C 180,E1 -16207.898,E2 -16207.898} C_VEL
LIN {X 0,Y 298.55,Z 192.797,A -85,B 0,C 180,E1 -16212.232,E2 -16212.232} C_VEL
LIN {X 0,Y 298.582,Z 192.791,A -85,B 0,C 180,E1 -16215.195,E2 -16215.195} C_VEL
LIN {X 0,Y 298.537,Z 192.797,A -85,B 0,C 180,E1 -16219.244,E2 -16219.244} C_VEL
LIN {X 0,Y 298.455,Z 192.812,A -85,B 0,C 180,E1 -16223.599,E2 -16223.599} C_VEL
LIN {X 0,Y 298.485,Z 192.803,A -85,B 0,C 180,E1 -16226.576,E2 -16226.576} C_VEL
LIN {X 0,Y 298.415,Z 192.817,A -85,B 0,C 180,E1 -16229.642,E2 -16229.642} C_VEL
LIN {X 0,Y 298.397,Z 192.818,A -85,B 0,C 180,E1 -16232.801,E2 -16232.801} C_VEL
LIN {X 0,Y 298.672,Z 194.562,A -85,B 0,C 180,E1 -16236.035,E2 -16236.035} C_VEL
LIN {X 0,Y 298.97,Z 196.781,A -85,B 0,C 180,E1 -16239.399,E2 -16239.399} C_VEL
LIN {X 0,Y 299.345,Z 199.314,A -85,B 0,C 180,E1 -16242.912,E2 -16242.912} C_VEL
LIN {X 0,Y 299.654,Z 202.245,A -85,B 0,C 180,E1 -16246.642,E2 -16246.642} C_VEL
LIN {X 0,Y 299.575,Z 204.213,A -85,B 0,C 180,E1 -16248.939,E2 -16248.939} C_VEL
LIN {X 0,Y 299.11,Z 207.318,A -85,B 0,C 180,E1 -16252.346,E2 -16252.346} C_VEL
LIN {X 0,Y 298.595,Z 210.466,A -85,B 0,C 180,E1 -16255.606,E2 -16255.606} C_VEL
LIN {X 0,Y 298.105,Z 213.637,A -85,B 0,C 180,E1 -16258.758,E2 -16258.758} C_VEL
LIN {X 0,Y 297.669,Z 216.825,A -85,B 0,C 180,E1 -16261.823,E2 -16261.823} C_VEL
LIN {X 0,Y 297.251,Z 220.677,A -85,B 0,C 180,E1 -16265.414,E2 -16265.414} C_VEL
LIN {X 0,Y 299.306,Z 228.602,A -85,B 0,C 180,E1 -16265.922,E2 -16265.922} C_VEL
LIN {X 0,Y 301.734,Z 239.217,A -85,B 0,C 180,E1 -16266.74,E2 -16266.74} C_VEL
LIN {X 0,Y 303.339,Z 248.938,A -85,B 0,C 180,E1 -16267.609,E2 -16267.609} C_VEL
LIN {X 0,Y 304.402,Z 257.581,A -85,B 0,C 180,E1 -16268.499,E2 -16268.499} C_VEL
LIN {X 0,Y 305.018,Z 266.917,A -85,B 0,C 180,E1 -16269.605,E2 -16269.605} C_VEL
LIN {X 0,Y 303.677,Z 275.862,A -85,B 0,C 180,E1 -16270.744,E2 -16270.744} C_VEL
LIN {X 0,Y 302.391,Z 284.396,A -85,B 0,C 180,E1 -16272.065,E2 -16272.065} C_VEL
LIN {X 0,Y 301.305,Z 291.571,A -85,B 0,C 180,E1 -16273.387,E2 -16273.387} C_VEL
LIN {X 0,Y 300.255,Z 297.823,A -85,B 0,C 180,E1 -16274.733,E2 -16274.733} C_VEL
LIN {X 0,Y 299.112,Z 304.362,A -85,B 0,C 180,E1 -16276.411,E2 -16276.411} C_VEL
LIN {X 0,Y 298.34,Z 308.865,A -85,B 0,C 180,E1 -16277.76,E2 -16277.76} C_VEL
LIN {X 0,Y 297.524,Z 314.361,A -85,B 0,C 180,E1 -16279.796,E2 -16279.796} C_VEL
LIN {X 0,Y 296.972,Z 318.691,A -85,B 0,C 180,E1 -16281.837,E2 -16281.837} C_VEL
LIN {X 0,Y 296.742,Z 321.061,A -85,B 0,C 180,E1 -16283.199,E2 -16283.199} C_VEL
LIN {X 0,Y 296.603,Z 322.863,A -85,B 0,C 180,E1 -16284.561,E2 -16284.561} C_VEL
LIN {X 0,Y 296.537,Z 325.315,A -85,B 0,C 180,E1 -16287.283,E2 -16287.283} C_VEL
LIN {X 0,Y 296.481,Z 325.904,A -85,B 0,C 180,E1 -16288.642,E2 -16288.642} C_VEL
LIN {X 0,Y 296.481,Z 325.904,A -85,B 0,C 180,E1 -16291.358,E2 -16291.358} C_VEL
LIN {X 0,Y 296.537,Z 325.315,A -85,B 0,C 180,E1 -16292.717,E2 -16292.717} C_VEL
LIN {X 0,Y 296.603,Z 322.863,A -85,B 0,C 180,E1 -16295.439,E2 -16295.439} C_VEL
LIN {X 0,Y 296.858,Z 319.91,A -85,B 0,C 180,E1 -16297.482,E2 -16297.482} C_VEL
LIN {X 0,Y 297.313,Z 315.917,A -85,B 0,C 180,E1 -16299.524,E2 -16299.524} C_VEL
LIN {X 0,Y 298.079,Z 310.784,A -85,B 0,C 180,E1 -16301.561,E2 -16301.561} C_VEL
LIN {X 0,Y 298.895,Z 305.518,A -85,B 0,C 180,E1 -16303.253,E2 -16303.253} C_VEL
LIN {X 0,Y 300.01,Z 299.2,A -85,B 0,C 180,E1 -16304.932,E2 -16304.932} C_VEL
LIN {X 0,Y 301.014,Z 293.246,A -85,B 0,C 180,E1 -16306.27,E2 -16306.27} C_VEL
LIN {X 0,Y 302.048,Z 286.314,A -85,B 0,C 180,E1 -16307.606,E2 -16307.606} C_VEL
LIN {X 0,Y 303.126,Z 279.266,A -85,B 0,C 180,E1 -16308.765,E2 -16308.765} C_VEL
LIN {X 0,Y 304.461,Z 270.973,A -85,B 0,C 180,E1 -16309.906,E2 -16309.906} C_VEL
LIN {X 0,Y 305.058,Z 265.561,A -85,B 0,C 180,E1 -16310.569,E2 -16310.569} C_VEL
LIN {X 0,Y 304.075,Z 254.366,A -85,B 0,C 180,E1 -16311.856,E2 -16311.856} C_VEL
LIN {X 0,Y 302.417,Z 242.939,A -85,B 0,C 180,E1 -16312.945,E2 -16312.945} C_VEL
LIN {X 0,Y 300.127,Z 231.982,A -85,B 0,C 180,E1 -16313.833,E2 -16313.833} C_VEL
LIN {X 0,Y 297.321,Z 221.317,A -85,B 0,C 180,E1 -16314.558,E2 -16314.558} C_VEL
LIN {X 0,Y 297.243,Z 220.62,A -85,B 0,C 180,E1 -16314.605,E2 -16314.605} C_VEL
LIN {X 0,Y 297.836,Z 215.757,A -85,B 0,C 180,E1 -16319.18,E2 -16319.18} C_VEL
LIN {X 0,Y 298.331,Z 212.028,A -85,B 0,C 180,E1 -16322.808,E2 -16322.808} C_VEL
LIN {X 0,Y 298.861,Z 208.884,A -85,B 0,C 180,E1 -16326.007,E2 -16326.007} C_VEL
LIN {X 0,Y 299.375,Z 205.758,A -85,B 0,C 180,E1 -16329.333,E2 -16329.333} C_VEL
LIN {X 0,Y 299.671,Z 202.651,A -85,B 0,C 180,E1 -16332.852,E2 -16332.852} C_VEL
LIN {X 0,Y 299.389,Z 199.596,A -85,B 0,C 180,E1 -16336.694,E2 -16336.694} C_VEL
LIN {X 0,Y 298.959,Z 196.763,A -85,B 0,C 180,E1 -16340.6,E2 -16340.6} C_VEL
LIN {X 0,Y 298.655,Z 194.567,A -85,B 0,C 180,E1 -16343.962,E2 -16343.962} C_VEL
LIN {X 0,Y 298.398,Z 192.819,A -85,B 0,C 180,E1 -16347.199,E2 -16347.199} C_VEL
LIN {X 0,Y 298.425,Z 192.814,A -85,B 0,C 180,E1 -16350.615,E2 -16350.615} C_VEL
LIN {X 0,Y 298.475,Z 192.805,A -85,B 0,C 180,E1 -16353.476,E2 -16353.476} C_VEL
LIN {X 0,Y 298.433,Z 192.814,A -85,B 0,C 180,E1 -16356.697,E2 -16356.697} C_VEL
LIN {X 0,Y 298.537,Z 192.798,A -85,B 0,C 180,E1 -16360.756,E2 -16360.756} C_VEL
LIN {X 0,Y 298.59,Z 192.789,A -85,B 0,C 180,E1 -16364.994,E2 -16364.994} C_VEL
LIN {X 0,Y 298.588,Z 192.79,A -85,B 0,C 180,E1 -16369.146,E2 -16369.146} C_VEL
LIN {X 0,Y 298.738,Z 192.775,A -85,B 0,C 180,E1 -16371.885,E2 -16371.885} C_VEL
LIN {X 0,Y 298.651,Z 192.782,A -85,B 0,C 180,E1 -16374.598,E2 -16374.598} C_VEL
LIN {X 0,Y 298.919,Z 192.746,A -85,B 0,C 180,E1 -16378.652,E2 -16378.652} C_VEL
LIN {X 0,Y 298.919,Z 192.742,A -85,B 0,C 180,E1 -16381.346,E2 -16381.346} C_VEL
LIN {X 0,Y 298.783,Z 192.765,A -85,B 0,C 180,E1 -16386.753,E2 -16386.753} C_VEL
LIN {X 0,Y 298.631,Z 192.785,A -85,B 0,C 180,E1 -16389.481,E2 -16389.481} C_VEL
LIN {X 0,Y 298.547,Z 192.795,A -85,B 0,C 180,E1 -16393.615,E2 -16393.615} C_VEL
LIN {X 0,Y 298.544,Z 192.794,A -85,B 0,C 180,E1 -16396.408,E2 -16396.408} C_VEL
LIN {X 0,Y 298.507,Z 192.797,A -85,B 0,C 180,E1 -16399.654,E2 -16399.654} C_VEL
LIN {X 0,Y 298.452,Z 192.806,A -85,B 0,C 180,E1 -16403.597,E2 -16403.597} C_VEL
LIN {X 0,Y 298.487,Z 192.803,A -85,B 0,C 180,E1 -16406.574,E2 -16406.574} C_VEL
LIN {X 0,Y 298.416,Z 192.811,A -85,B 0,C 180,E1 -16409.641,E2 -16409.641} C_VEL
LIN {X 0,Y 298.39,Z 192.818,A -85,B 0,C 180,E1 -16412.8,E2 -16412.8} C_VEL
LIN {X 0,Y 298.46,Z 192.808,A -85,B 0,C 180,E1 -16416.812,E2 -16416.812} C_VEL
LIN {X 0,Y 298.412,Z 192.812,A -85,B 0,C 180,E1 -16421.094,E2 -16421.094} C_VEL
LIN {X 0,Y 298.421,Z 192.811,A -85,B 0,C 180,E1 -16423.109,E2 -16423.109} C_VEL
LIN {X 0,Y 298.398,Z 192.813,A -85,B 0,C 180,E1 -16426.921,E2 -16426.921} C_VEL
LIN {X 0,Y 298.41,Z 192.812,A -85,B 0,C 180,E1 -16431.004,E2 -16431.004} C_VEL
LIN {X 0,Y 298.416,Z 192.815,A -85,B 0,C 180,E1 -16433.93,E2 -16433.93} C_VEL
LIN {X 0,Y 298.395,Z 192.818,A -85,B 0,C 180,E1 -16437.982,E2 -16437.982} C_VEL
LIN {X 0,Y 298.472,Z 192.808,A -85,B 0,C 180,E1 -16441.906,E2 -16441.906} C_VEL
LIN {X 0,Y 298.465,Z 192.807,A -85,B 0,C 180,E1 -16445.156,E2 -16445.156} C_VEL
LIN {X 0,Y 299.497,Z 195.707,A -85,B 0,C 180,E1 -16445.338,E2 -16445.338} C_VEL
LIN {X 0,Y 303.205,Z 202.99,A -85,B 0,C 180,E1 -16445.869,E2 -16445.869} C_VEL
LIN {X 0,Y 307.502,Z 210.087,A -85,B 0,C 180,E1 -16446.498,E2 -16446.498} C_VEL
LIN {X 0,Y 313.492,Z 218.209,A -85,B 0,C 180,E1 -16447.435,E2 -16447.435} C_VEL
LIN {X 0,Y 320.385,Z 226.799,A -85,B 0,C 180,E1 -16448.664,E2 -16448.664} C_VEL
LIN {X 0,Y 327.155,Z 234.605,A -85,B 0,C 180,E1 -16450.023,E2 -16450.023} C_VEL
LIN {X 0,Y 332.117,Z 240.002,A -85,B 0,C 180,E1 -16451.11,E2 -16451.11} C_VEL
LIN {X 0,Y 339.676,Z 247.808,A -85,B 0,C 180,E1 -16452.94,E2 -16452.94} C_VEL
LIN {X 0,Y 345.084,Z 252.914,A -85,B 0,C 180,E1 -16454.388,E2 -16454.388} C_VEL
LIN {X 0,Y 348.516,Z 256.46,A -85,B 0,C 180,E1 -16455.45,E2 -16455.45} C_VEL
LIN {X 0,Y 353.4,Z 260.695,A -85,B 0,C 180,E1 -16457.018,E2 -16457.018} C_VEL
LIN {X 0,Y 358.198,Z 265.07,A -85,B 0,C 180,E1 -16458.816,E2 -16458.816} C_VEL
LIN {X 0,Y 361.101,Z 266.925,A -85,B 0,C 180,E1 -16459.912,E2 -16459.912} C_VEL
LIN {X 0,Y 363.344,Z 269.236,A -85,B 0,C 180,E1 -16461.098,E2 -16461.098} C_VEL
LIN {X 0,Y 365.277,Z 271.217,A -85,B 0,C 180,E1 -16462.26,E2 -16462.26} C_VEL
LIN {X 0,Y 367.604,Z 273.068,A -85,B 0,C 180,E1 -16463.797,E2 -16463.797} C_VEL
LIN {X 0,Y 370.002,Z 274.394,A -85,B 0,C 180,E1 -16465.643,E2 -16465.643} C_VEL
LIN {X 0,Y 371.195,Z 274.772,A -85,B 0,C 180,E1 -16466.744,E2 -16466.744} C_VEL
LIN {X 0,Y 372.566,Z 275.078,A -85,B 0,C 180,E1 -16468.761,E2 -16468.761} C_VEL
LIN {X 0,Y 372.806,Z 275.147,A -85,B 0,C 180,E1 -16470,E2 -16470} C_VEL
LIN {X 0,Y 372.565,Z 275.071,A -85,B 0,C 180,E1 -16471.23,E2 -16471.23} C_VEL
LIN {X 0,Y 371.186,Z 274.763,A -85,B 0,C 180,E1 -16473.256,E2 -16473.256} C_VEL
LIN {X 0,Y 370.003,Z 274.396,A -85,B 0,C 180,E1 -16474.357,E2 -16474.357} C_VEL
LIN {X 0,Y 367.618,Z 273.017,A -85,B 0,C 180,E1 -16476.224,E2 -16476.224} C_VEL
LIN {X 0,Y 365.287,Z 271.193,A -85,B 0,C 180,E1 -16477.74,E2 -16477.74} C_VEL
LIN {X 0,Y 362.999,Z 268.831,A -85,B 0,C 180,E1 -16479.107,E2 -16479.107} C_VEL
LIN {X 0,Y 361.047,Z 266.974,A -85,B 0,C 180,E1 -16480.09,E2 -16480.09} C_VEL
LIN {X 0,Y 356.301,Z 263.483,A -85,B 0,C 180,E1 -16481.903,E2 -16481.903} C_VEL
LIN {X 0,Y 351.935,Z 259.292,A -85,B 0,C 180,E1 -16483.496,E2 -16483.496} C_VEL
LIN {X 0,Y 347.274,Z 255.222,A -85,B 0,C 180,E1 -16484.944,E2 -16484.944} C_VEL
LIN {X 0,Y 342.285,Z 250.272,A -85,B 0,C 180,E1 -16486.395,E2 -16486.395} C_VEL
LIN {X 0,Y 336.307,Z 244.257,A -85,B 0,C 180,E1 -16487.915,E2 -16487.915} C_VEL
LIN {X 0,Y 330.631,Z 238.22,A -85,B 0,C 180,E1 -16489.248,E2 -16489.248} C_VEL
LIN {X 0,Y 326.278,Z 233.637,A -85,B 0,C 180,E1 -16490.159,E2 -16490.159} C_VEL
LIN {X 0,Y 319.562,Z 225.704,A -85,B 0,C 180,E1 -16491.501,E2 -16491.501} C_VEL
LIN {X 0,Y 312.255,Z 216.699,A -85,B 0,C 180,E1 -16492.768,E2 -16492.768} C_VEL
LIN {X 0,Y 306.485,Z 208.413,A -85,B 0,C 180,E1 -16493.654,E2 -16493.654} C_VEL
LIN {X 0,Y 301.866,Z 200.745,A -85,B 0,C 180,E1 -16494.317,E2 -16494.317} C_VEL
LIN {X 0,Y 298.574,Z 193.481,A -85,B 0,C 180,E1 -16494.802,E2 -16494.802} C_VEL
LIN {X 0,Y 298.475,Z 192.806,A -85,B 0,C 180,E1 -16494.877,E2 -16494.877} C_VEL
LIN {X 0,Y 298.472,Z 192.808,A -85,B 0,C 180,E1 -16498.094,E2 -16498.094} C_VEL
LIN {X 0,Y 298.395,Z 192.818,A -85,B 0,C 180,E1 -16502.018,E2 -16502.018} C_VEL
LIN {X 0,Y 298.43,Z 192.813,A -85,B 0,C 180,E1 -16506.068,E2 -16506.068} C_VEL
LIN {X 0,Y 298.415,Z 192.813,A -85,B 0,C 180,E1 -16509.484,E2 -16509.484} C_VEL
LIN {X 0,Y 298.421,Z 192.81,A -85,B 0,C 180,E1 -16513.109,E2 -16513.109} C_VEL
LIN {X 0,Y 298.398,Z 192.814,A -85,B 0,C 180,E1 -16516.921,E2 -16516.921} C_VEL
LIN {X 0,Y 298.421,Z 192.812,A -85,B 0,C 180,E1 -16521.001,E2 -16521.001} C_VEL
LIN {X 0,Y 298.427,Z 192.81,A -85,B 0,C 180,E1 -16523.932,E2 -16523.932} C_VEL
LIN {X 0,Y 298.39,Z 192.814,A -85,B 0,C 180,E1 -16527.984,E2 -16527.984} C_VEL
LIN {X 0,Y 298.465,Z 192.805,A -85,B 0,C 180,E1 -16531.905,E2 -16531.905} C_VEL
LIN {X 0,Y 298.481,Z 192.804,A -85,B 0,C 180,E1 -16534.924,E2 -16534.924} C_VEL
LIN {X 0,Y 298.445,Z 192.806,A -85,B 0,C 180,E1 -16539.316,E2 -16539.316} C_VEL
LIN {X 0,Y 298.533,Z 192.797,A -85,B 0,C 180,E1 -16542.18,E2 -16542.18} C_VEL
LIN {X 0,Y 298.588,Z 192.791,A -85,B 0,C 180,E1 -16544.995,E2 -16544.995} C_VEL
LIN {X 0,Y 298.587,Z 192.789,A -85,B 0,C 180,E1 -16549.147,E2 -16549.147} C_VEL
LIN {X 0,Y 298.736,Z 192.771,A -85,B 0,C 180,E1 -16551.886,E2 -16551.886} C_VEL
LIN {X 0,Y 298.652,Z 192.782,A -85,B 0,C 180,E1 -16554.6,E2 -16554.6} C_VEL
LIN {X 0,Y 298.919,Z 192.742,A -85,B 0,C 180,E1 -16558.654,E2 -16558.654} C_VEL
LIN {X 0,Y 298.919,Z 192.746,A -85,B 0,C 180,E1 -16561.348,E2 -16561.348} C_VEL
LIN {X 0,Y 298.783,Z 192.766,A -85,B 0,C 180,E1 -16566.755,E2 -16566.755} C_VEL
LIN {X 0,Y 298.733,Z 192.774,A -85,B 0,C 180,E1 -16567.898,E2 -16567.898} C_VEL
LIN {X 0,Y 298.051,Z 192.863,A -85,B 0,C 180,E1 -16569.022,E2 -16569.022} C_VEL
LIN {X 0,Y 295.097,Z 193.228,A -85,B 0,C 180,E1 -16570.849,E2 -16570.849} C_VEL
LIN {X 0,Y 292.61,Z 193.536,A -85,B 0,C 180,E1 -16572.331,E2 -16572.331} C_VEL
LIN {X 0,Y 291.578,Z 193.665,A -85,B 0,C 180,E1 -16573.482,E2 -16573.482} C_VEL
LIN {X 0,Y 291.514,Z 193.674,A -85,B 0,C 180,E1 -16573.873,E2 -16573.873} C_VEL
LIN {X 0,Y 291.484,Z 193.675,A -85,B 0,C 180,E1 -16576.819,E2 -16576.819} C_VEL
LIN {X 0,Y 291.449,Z 193.683,A -85,B 0,C 180,E1 -16579.876,E2 -16579.876} C_VEL
LIN {X 0,Y 291.398,Z 193.686,A -85,B 0,C 180,E1 -16584.206,E2 -16584.206} C_VEL
LIN {X 0,Y 291.418,Z 193.686,A -85,B 0,C 180,E1 -16587.273,E2 -16587.273} C_VEL
LIN {X 0,Y 291.333,Z 193.697,A -85,B 0,C 180,E1 -16590.438,E2 -16590.438} C_VEL
LIN {X 0,Y 291.343,Z 193.698,A -85,B 0,C 180,E1 -16592.405,E2 -16592.405} C_VEL
LIN {X 0,Y 291.603,Z 195.249,A -85,B 0,C 180,E1 -16595.341,E2 -16595.341} C_VEL
LIN {X 0,Y 291.963,Z 198.003,A -85,B 0,C 180,E1 -16599.621,E2 -16599.621} C_VEL
LIN {X 0,Y 292.259,Z 199.887,A -85,B 0,C 180,E1 -16602.325,E2 -16602.325} C_VEL
LIN {X 0,Y 292.572,Z 202.765,A -85,B 0,C 180,E1 -16606.109,E2 -16606.109} C_VEL
LIN {X 0,Y 292.442,Z 205.634,A -85,B 0,C 180,E1 -16609.544,E2 -16609.544} C_VEL
LIN {X 0,Y 291.961,Z 208.744,A -85,B 0,C 180,E1 -16613.002,E2 -16613.002} C_VEL
LIN {X 0,Y 291.387,Z 211.883,A -85,B 0,C 180,E1 -16616.308,E2 -16616.308} C_VEL
LIN {X 0,Y 290.79,Z 216.01,A -85,B 0,C 180,E1 -16620.468,E2 -16620.468} C_VEL
LIN {X 0,Y 290.241,Z 220.436,A -85,B 0,C 180,E1 -16624.773,E2 -16624.773} C_VEL
LIN {X 0,Y 292.15,Z 227.782,A -85,B 0,C 180,E1 -16625.261,E2 -16625.261} C_VEL
LIN {X 0,Y 294.776,Z 238.947,A -85,B 0,C 180,E1 -16626.154,E2 -16626.154} C_VEL
LIN {X 0,Y 296.278,Z 247.479,A -85,B 0,C 180,E1 -16626.933,E2 -16626.933} C_VEL
LIN {X 0,Y 297.562,Z 257.963,A -85,B 0,C 180,E1 -16628.046,E2 -16628.046} C_VEL
LIN {X 0,Y 298.259,Z 266.715,A -85,B 0,C 180,E1 -16629.123,E2 -16629.123} C_VEL
LIN {X 0,Y 296.981,Z 275.651,A -85,B 0,C 180,E1 -16630.292,E2 -16630.292} C_VEL
LIN {X 0,Y 295.602,Z 284.183,A -85,B 0,C 180,E1 -16631.638,E2 -16631.638} C_VEL
LIN {X 0,Y 294.607,Z 290.383,A -85,B 0,C 180,E1 -16632.784,E2 -16632.784} C_VEL
LIN {X 0,Y 293.358,Z 297.61,A -85,B 0,C 180,E1 -16634.365,E2 -16634.365} C_VEL
LIN {X 0,Y 292.189,Z 304.15,A -85,B 0,C 180,E1 -16636.082,E2 -16636.082} C_VEL
LIN {X 0,Y 291.37,Z 308.653,A -85,B 0,C 180,E1 -16637.462,E2 -16637.462} C_VEL
LIN {X 0,Y 290.515,Z 314.149,A -85,B 0,C 180,E1 -16639.547,E2 -16639.547} C_VEL
LIN {X 0,Y 289.916,Z 318.478,A -85,B 0,C 180,E1 -16641.637,E2 -16641.637} C_VEL
LIN {X 0,Y 289.669,Z 320.849,A -85,B 0,C 180,E1 -16643.032,E2 -16643.032} C_VEL
LIN {X 0,Y 289.519,Z 322.651,A -85,B 0,C 180,E1 -16644.428,E2 -16644.428} C_VEL
LIN {X 0,Y 289.443,Z 325.103,A -85,B 0,C 180,E1 -16647.217,E2 -16647.217} C_VEL
LIN {X 0,Y 289.404,Z 325.693,A -85,B 0,C 180,E1 -16648.608,E2 -16648.608} C_VEL
LIN {X 0,Y 289.404,Z 325.693,A -85,B 0,C 180,E1 -16651.392,E2 -16651.392} C_VEL
LIN {X 0,Y 289.443,Z 325.103,A -85,B 0,C 180,E1 -16652.783,E2 -16652.783} C_VEL
LIN {X 0,Y 289.519,Z 322.651,A -85,B 0,C 180,E1 -16655.572,E2 -16655.572} C_VEL
LIN {X 0,Y 289.81,Z 319.698,A -85,B 0,C 180,E1 -16657.665,E2 -16657.665} C_VEL
LIN {X 0,Y 290.294,Z 315.705,A -85,B 0,C 180,E1 -16659.757,E2 -16659.757} C_VEL
LIN {X 0,Y 291.077,Z 310.571,A -85,B 0,C 180,E1 -16661.843,E2 -16661.843} C_VEL
LIN {X 0,Y 291.968,Z 305.306,A -85,B 0,C 180,E1 -16663.573,E2 -16663.573} C_VEL
LIN {X 0,Y 293.117,Z 298.987,A -85,B 0,C 180,E1 -16665.292,E2 -16665.292} C_VEL
LIN {X 0,Y 294.196,Z 293.035,A -85,B 0,C 180,E1 -16666.658,E2 -16666.658} C_VEL
LIN {X 0,Y 295.265,Z 286.102,A -85,B 0,C 180,E1 -16668.025,E2 -16668.025} C_VEL
LIN {X 0,Y 296.581,Z 277.92,A -85,B 0,C 180,E1 -16669.375,E2 -16669.375} C_VEL
LIN {X 0,Y 297.937,Z 269.409,A -85,B 0,C 180,E1 -16670.541,E2 -16670.541} C_VEL
LIN {X 0,Y 298.16,Z 265.364,A -85,B 0,C 180,E1 -16671.064,E2 -16671.064} C_VEL
LIN {X 0,Y 297.174,Z 253.987,A -85,B 0,C 180,E1 -16672.405,E2 -16672.405} C_VEL
LIN {X 0,Y 295.517,Z 242.769,A -85,B 0,C 180,E1 -16673.509,E2 -16673.509} C_VEL
LIN {X 0,Y 293.154,Z 231.754,A -85,B 0,C 180,E1 -16674.436,E2 -16674.436} C_VEL
LIN {X 0,Y 290.364,Z 221.64,A -85,B 0,C 180,E1 -16675.167,E2 -16675.167} C_VEL
LIN {X 0,Y 290.238,Z 220.436,A -85,B 0,C 180,E1 -16675.227,E2 -16675.227} C_VEL
LIN {X 0,Y 290.787,Z 215.996,A -85,B 0,C 180,E1 -16679.531,E2 -16679.531} C_VEL
LIN {X 0,Y 291.387,Z 211.877,A -85,B 0,C 180,E1 -16683.692,E2 -16683.692} C_VEL
LIN {X 0,Y 292.009,Z 208.355,A -85,B 0,C 180,E1 -16687.416,E2 -16687.416} C_VEL
LIN {X 0,Y 292.44,Z 205.62,A -85,B 0,C 180,E1 -16690.456,E2 -16690.456} C_VEL
LIN {X 0,Y 292.572,Z 202.738,A -85,B 0,C 180,E1 -16693.891,E2 -16693.891} C_VEL
LIN {X 0,Y 292.246,Z 199.878,A -85,B 0,C 180,E1 -16697.673,E2 -16697.673} C_VEL
LIN {X 0,Y 291.859,Z 197.414,A -85,B 0,C 180,E1 -16701.237,E2 -16701.237} C_VEL
LIN {X 0,Y 291.575,Z 195.026,A -85,B 0,C 180,E1 -16705.036,E2 -16705.036} C_VEL
LIN {X 0,Y 291.37,Z 193.692,A -85,B 0,C 180,E1 -16707.95,E2 -16707.95} C_VEL
LIN {X 0,Y 291.375,Z 193.691,A -85,B 0,C 180,E1 -16711.157,E2 -16711.157} C_VEL
LIN {X 0,Y 291.411,Z 193.69,A -85,B 0,C 180,E1 -16714.271,E2 -16714.271} C_VEL
LIN {X 0,Y 291.387,Z 193.689,A -85,B 0,C 180,E1 -16717.299,E2 -16717.299} C_VEL
LIN {X 0,Y 291.456,Z 193.684,A -85,B 0,C 180,E1 -16720.269,E2 -16720.269} C_VEL
LIN {X 0,Y 291.538,Z 193.669,A -85,B 0,C 180,E1 -16724.634,E2 -16724.634} C_VEL
LIN {X 0,Y 291.532,Z 193.669,A -85,B 0,C 180,E1 -16728.88,E2 -16728.88} C_VEL
LIN {X 0,Y 291.684,Z 193.652,A -85,B 0,C 180,E1 -16731.687,E2 -16731.687} C_VEL
LIN {X 0,Y 291.622,Z 193.658,A -85,B 0,C 180,E1 -16734.467,E2 -16734.467} C_VEL
LIN {X 0,Y 291.885,Z 193.623,A -85,B 0,C 180,E1 -16738.62,E2 -16738.62} C_VEL
LIN {X 0,Y 291.885,Z 193.617,A -85,B 0,C 180,E1 -16741.379,E2 -16741.379} C_VEL
LIN {X 0,Y 291.731,Z 193.644,A -85,B 0,C 180,E1 -16746.917,E2 -16746.917} C_VEL
LIN {X 0,Y 291.57,Z 193.664,A -85,B 0,C 180,E1 -16749.713,E2 -16749.713} C_VEL
LIN {X 0,Y 291.517,Z 193.669,A -85,B 0,C 180,E1 -16753.95,E2 -16753.95} C_VEL
LIN {X 0,Y 291.482,Z 193.676,A -85,B 0,C 180,E1 -16756.817,E2 -16756.817} C_VEL
LIN {X 0,Y 291.446,Z 193.676,A -85,B 0,C 180,E1 -16759.874,E2 -16759.874} C_VEL
LIN {X 0,Y 291.395,Z 193.684,A -85,B 0,C 180,E1 -16764.205,E2 -16764.205} C_VEL
LIN {X 0,Y 291.421,Z 193.684,A -85,B 0,C 180,E1 -16767.271,E2 -16767.271} C_VEL
LIN {X 0,Y 291.332,Z 193.696,A -85,B 0,C 180,E1 -16770.436,E2 -16770.436} C_VEL
LIN {X 0,Y 291.34,Z 193.692,A -85,B 0,C 180,E1 -16773.698,E2 -16773.698} C_VEL
LIN {X 0,Y 291.393,Z 193.686,A -85,B 0,C 180,E1 -16777.259,E2 -16777.259} C_VEL
LIN {X 0,Y 291.371,Z 193.692,A -85,B 0,C 180,E1 -16780.635,E2 -16780.635} C_VEL
LIN {X 0,Y 291.294,Z 193.702,A -85,B 0,C 180,E1 -16784.4,E2 -16784.4} C_VEL
LIN {X 0,Y 291.321,Z 193.698,A -85,B 0,C 180,E1 -16788.404,E2 -16788.404} C_VEL
LIN {X 0,Y 291.359,Z 193.69,A -85,B 0,C 180,E1 -16791.16,E2 -16791.16} C_VEL
LIN {X 0,Y 291.357,Z 193.692,A -85,B 0,C 180,E1 -16794.626,E2 -16794.626} C_VEL
LIN {X 0,Y 291.371,Z 193.693,A -85,B 0,C 180,E1 -16797.951,E2 -16797.951} C_VEL
LIN {X 0,Y 291.386,Z 193.688,A -85,B 0,C 180,E1 -16801.159,E2 -16801.159} C_VEL
LIN {X 0,Y 291.442,Z 193.682,A -85,B 0,C 180,E1 -16804.542,E2 -16804.542} C_VEL
LIN {X 0,Y 292.361,Z 196.419,A -85,B 0,C 180,E1 -16804.707,E2 -16804.707} C_VEL
LIN {X 0,Y 297.571,Z 206.949,A -85,B 0,C 180,E1 -16805.518,E2 -16805.518} C_VEL
LIN {X 0,Y 302.24,Z 214.715,A -85,B 0,C 180,E1 -16806.287,E2 -16806.287} C_VEL
LIN {X 0,Y 308.22,Z 222.883,A -85,B 0,C 180,E1 -16807.268,E2 -16807.268} C_VEL
LIN {X 0,Y 315.319,Z 231.723,A -85,B 0,C 180,E1 -16808.539,E2 -16808.539} C_VEL
LIN {X 0,Y 321.88,Z 239.292,A -85,B 0,C 180,E1 -16809.86,E2 -16809.86} C_VEL
LIN {X 0,Y 328.26,Z 246.22,A -85,B 0,C 180,E1 -16811.268,E2 -16811.268} C_VEL
LIN {X 0,Y 334.944,Z 253.09,A -85,B 0,C 180,E1 -16812.917,E2 -16812.917} C_VEL
LIN {X 0,Y 340.625,Z 258.523,A -85,B 0,C 180,E1 -16814.442,E2 -16814.442} C_VEL
LIN {X 0,Y 345.275,Z 262.935,A -85,B 0,C 180,E1 -16815.862,E2 -16815.862} C_VEL
LIN {X 0,Y 350.248,Z 267.566,A -85,B 0,C 180,E1 -16817.572,E2 -16817.572} C_VEL
LIN {X 0,Y 354.375,Z 270.986,A -85,B 0,C 180,E1 -16819.134,E2 -16819.134} C_VEL
LIN {X 0,Y 356.733,Z 272.578,A -85,B 0,C 180,E1 -16820.076,E2 -16820.076} C_VEL
LIN {X 0,Y 360.385,Z 276.317,A -85,B 0,C 180,E1 -16822.154,E2 -16822.154} C_VEL
LIN {X 0,Y 362.177,Z 277.842,A -85,B 0,C 180,E1 -16823.314,E2 -16823.314} C_VEL
LIN {X 0,Y 363.789,Z 278.944,A -85,B 0,C 180,E1 -16824.457,E2 -16824.457} C_VEL
LIN {X 0,Y 366.169,Z 280.045,A -85,B 0,C 180,E1 -16826.413,E2 -16826.413} C_VEL
LIN {X 0,Y 367.405,Z 280.41,A -85,B 0,C 180,E1 -16827.808,E2 -16827.808} C_VEL
LIN {X 0,Y 368.051,Z 280.482,A -85,B 0,C 180,E1 -16828.906,E2 -16828.906} C_VEL
LIN {X 0,Y 368.211,Z 280.555,A -85,B 0,C 180,E1 -16830,E2 -16830} C_VEL
LIN {X 0,Y 368.047,Z 280.469,A -85,B 0,C 180,E1 -16831.094,E2 -16831.094} C_VEL
LIN {X 0,Y 367.404,Z 280.39,A -85,B 0,C 180,E1 -16832.193,E2 -16832.193} C_VEL
LIN {X 0,Y 366.174,Z 280.023,A -85,B 0,C 180,E1 -16833.601,E2 -16833.601} C_VEL
LIN {X 0,Y 363.807,Z 278.962,A -85,B 0,C 180,E1 -16835.543,E2 -16835.543} C_VEL
LIN {X 0,Y 361.328,Z 277.103,A -85,B 0,C 180,E1 -16837.27,E2 -16837.27} C_VEL
LIN {X 0,Y 358.446,Z 274.296,A -85,B 0,C 180,E1 -16839.024,E2 -16839.024} C_VEL
LIN {X 0,Y 356.002,Z 272.078,A -85,B 0,C 180,E1 -16840.234,E2 -16840.234} C_VEL
LIN {X 0,Y 351.839,Z 269.007,A -85,B 0,C 180,E1 -16841.829,E2 -16841.829} C_VEL
LIN {X 0,Y 347.033,Z 264.434,A -85,B 0,C 180,E1 -16843.574,E2 -16843.574} C_VEL
LIN {X 0,Y 342.126,Z 260.071,A -85,B 0,C 180,E1 -16845.102,E2 -16845.102} C_VEL
LIN {X 0,Y 337.197,Z 255.218,A -85,B 0,C 180,E1 -16846.517,E2 -16846.517} C_VEL
LIN {X 0,Y 329.635,Z 247.612,A -85,B 0,C 180,E1 -16848.425,E2 -16848.425} C_VEL
LIN {X 0,Y 321.892,Z 239.317,A -85,B 0,C 180,E1 -16850.145,E2 -16850.145} C_VEL
LIN {X 0,Y 315.308,Z 231.7,A -85,B 0,C 180,E1 -16851.458,E2 -16851.458} C_VEL
LIN {X 0,Y 308.224,Z 222.854,A -85,B 0,C 180,E1 -16852.734,E2 -16852.734} C_VEL
LIN {X 0,Y 301.378,Z 213.33,A -85,B 0,C 180,E1 -16853.858,E2 -16853.858} C_VEL
LIN {X 0,Y 296.709,Z 205.44,A -85,B 0,C 180,E1 -16854.621,E2 -16854.621} C_VEL
LIN {X 0,Y 291.631,Z 194.72,A -85,B 0,C 180,E1 -16855.407,E2 -16855.407} C_VEL
LIN {X 0,Y 291.445,Z 193.681,A -85,B 0,C 180,E1 -16855.486,E2 -16855.486} C_VEL
LIN {X 0,Y 291.386,Z 193.69,A -85,B 0,C 180,E1 -16859.741,E2 -16859.741} C_VEL
LIN {X 0,Y 291.341,Z 193.695,A -85,B 0,C 180,E1 -16863.698,E2 -16863.698} C_VEL
LIN {X 0,Y 291.4,Z 193.686,A -85,B 0,C 180,E1 -16867.261,E2 -16867.261} C_VEL
LIN {X 0,Y 291.372,Z 193.688,A -85,B 0,C 180,E1 -16870.635,E2 -16870.635} C_VEL
LIN {X 0,Y 291.293,Z 193.698,A -85,B 0,C 180,E1 -16874.4,E2 -16874.4} C_VEL
LIN {X 0,Y 291.345,Z 193.692,A -85,B 0,C 180,E1 -16878.399,E2 -16878.399} C_VEL
LIN {X 0,Y 291.37,Z 193.691,A -85,B 0,C 180,E1 -16881.162,E2 -16881.162} C_VEL
LIN {X 0,Y 291.38,Z 193.687,A -85,B 0,C 180,E1 -16884.63,E2 -16884.63} C_VEL
LIN {X 0,Y 291.366,Z 193.689,A -85,B 0,C 180,E1 -16887.951,E2 -16887.951} C_VEL
LIN {X 0,Y 291.38,Z 193.691,A -85,B 0,C 180,E1 -16891.159,E2 -16891.159} C_VEL
LIN {X 0,Y 291.415,Z 193.682,A -85,B 0,C 180,E1 -16894.273,E2 -16894.273} C_VEL
LIN {X 0,Y 291.376,Z 193.69,A -85,B 0,C 180,E1 -16897.3,E2 -16897.3} C_VEL
LIN {X 0,Y 291.453,Z 193.675,A -85,B 0,C 180,E1 -16900.271,E2 -16900.271} C_VEL
LIN {X 0,Y 291.551,Z 193.668,A -85,B 0,C 180,E1 -16904.624,E2 -16904.624} C_VEL
LIN {X 0,Y 291.531,Z 193.669,A -85,B 0,C 180,E1 -16908.881,E2 -16908.881} C_VEL
LIN {X 0,Y 291.683,Z 193.649,A -85,B 0,C 180,E1 -16911.689,E2 -16911.689} C_VEL
LIN {X 0,Y 291.622,Z 193.659,A -85,B 0,C 180,E1 -16914.469,E2 -16914.469} C_VEL
LIN {X 0,Y 291.885,Z 193.617,A -85,B 0,C 180,E1 -16918.621,E2 -16918.621} C_VEL
LIN {X 0,Y 291.885,Z 193.623,A -85,B 0,C 180,E1 -16921.38,E2 -16921.38} C_VEL
LIN {X 0,Y 291.731,Z 193.644,A -85,B 0,C 180,E1 -16926.919,E2 -16926.919} C_VEL
LIN {X 0,Y 291.572,Z 193.666,A -85,B 0,C 180,E1 -16929.715,E2 -16929.715} C_VEL
LIN {X 0,Y 291.514,Z 193.674,A -85,B 0,C 180,E1 -16933.873,E2 -16933.873} C_VEL
LIN {X 0,Y 290.879,Z 193.759,A -85,B 0,C 180,E1 -16935.025,E2 -16935.025} C_VEL
LIN {X 0,Y 287.971,Z 194.117,A -85,B 0,C 180,E1 -16936.9,E2 -16936.9} C_VEL
LIN {X 0,Y 285.492,Z 194.422,A -85,B 0,C 180,E1 -16938.422,E2 -16938.422} C_VEL
LIN {X 0,Y 284.452,Z 194.554,A -85,B 0,C 180,E1 -16939.603,E2 -16939.603} C_VEL
LIN {X 0,Y 284.382,Z 194.561,A -85,B 0,C 180,E1 -16940.004,E2 -16940.004} C_VEL
LIN {X 0,Y 284.367,Z 194.564,A -85,B 0,C 180,E1 -16943.876,E2 -16943.876} C_VEL
LIN {X 0,Y 284.394,Z 194.561,A -85,B 0,C 180,E1 -16947.174,E2 -16947.174} C_VEL
LIN {X 0,Y 284.293,Z 194.577,A -85,B 0,C 180,E1 -16951.275,E2 -16951.275} C_VEL
LIN {X 0,Y 284.358,Z 195.001,A -85,B 0,C 180,E1 -16952.939,E2 -16952.939} C_VEL
LIN {X 0,Y 284.651,Z 196.954,A -85,B 0,C 180,E1 -16956.34,E2 -16956.34} C_VEL
LIN {X 0,Y 284.992,Z 199.386,A -85,B 0,C 180,E1 -16960.141,E2 -16960.141} C_VEL
LIN {X 0,Y 285.34,Z 201.81,A -85,B 0,C 180,E1 -16963.603,E2 -16963.603} C_VEL
LIN {X 0,Y 285.536,Z 203.966,A -85,B 0,C 180,E1 -16966.436,E2 -16966.436} C_VEL
LIN {X 0,Y 285.38,Z 206.699,A -85,B 0,C 180,E1 -16969.769,E2 -16969.769} C_VEL
LIN {X 0,Y 284.748,Z 210.152,A -85,B 0,C 180,E1 -16973.676,E2 -16973.676} C_VEL
LIN {X 0,Y 284.16,Z 213.483,A -85,B 0,C 180,E1 -16977.237,E2 -16977.237} C_VEL
LIN {X 0,Y 283.725,Z 216.453,A -85,B 0,C 180,E1 -16980.304,E2 -16980.304} C_VEL
LIN {X 0,Y 283.245,Z 220.408,A -85,B 0,C 180,E1 -16984.118,E2 -16984.118} C_VEL
LIN {X 0,Y 285.188,Z 227.846,A -85,B 0,C 180,E1 -16984.631,E2 -16984.631} C_VEL
LIN {X 0,Y 287.641,Z 237.818,A -85,B 0,C 180,E1 -16985.458,E2 -16985.458} C_VEL
LIN {X 0,Y 289.485,Z 247.717,A -85,B 0,C 180,E1 -16986.402,E2 -16986.402} C_VEL
LIN {X 0,Y 290.711,Z 257.723,A -85,B 0,C 180,E1 -16987.499,E2 -16987.499} C_VEL
LIN {X 0,Y 291.367,Z 266.598,A -85,B 0,C 180,E1 -16988.619,E2 -16988.619} C_VEL
LIN {X 0,Y 291.128,Z 270.55,A -85,B 0,C 180,E1 -16989.141,E2 -16989.141} C_VEL
LIN {X 0,Y 289.154,Z 282.05,A -85,B 0,C 180,E1 -16990.845,E2 -16990.845} C_VEL
LIN {X 0,Y 287.68,Z 290.853,A -85,B 0,C 180,E1 -16992.51,E2 -16992.51} C_VEL
LIN {X 0,Y 286.475,Z 297.397,A -85,B 0,C 180,E1 -16993.979,E2 -16993.979} C_VEL
LIN {X 0,Y 285.269,Z 303.938,A -85,B 0,C 180,E1 -16995.738,E2 -16995.738} C_VEL
LIN {X 0,Y 284.41,Z 308.44,A -85,B 0,C 180,E1 -16997.15,E2 -16997.15} C_VEL
LIN {X 0,Y 283.52,Z 313.938,A -85,B 0,C 180,E1 -16999.286,E2 -16999.286} C_VEL
LIN {X 0,Y 282.881,Z 318.267,A -85,B 0,C 180,E1 -17001.427,E2 -17001.427} C_VEL
LIN {X 0,Y 282.597,Z 320.637,A -85,B 0,C 180,E1 -17002.857,E2 -17002.857} C_VEL
LIN {X 0,Y 282.432,Z 322.682,A -85,B 0,C 180,E1 -17004.481,E2 -17004.481} C_VEL
LIN {X 0,Y 282.351,Z 324.892,A -85,B 0,C 180,E1 -17007.147,E2 -17007.147} C_VEL
LIN {X 0,Y 282.328,Z 325.482,A -85,B 0,C 180,E1 -17008.574,E2 -17008.574} C_VEL
LIN {X 0,Y 282.328,Z 325.482,A -85,B 0,C 180,E1 -17011.426,E2 -17011.426} C_VEL
LIN {X 0,Y 282.351,Z 324.892,A -85,B 0,C 180,E1 -17012.853,E2 -17012.853} C_VEL
LIN {X 0,Y 282.444,Z 322.439,A -85,B 0,C 180,E1 -17015.712,E2 -17015.712} C_VEL
LIN {X 0,Y 282.744,Z 319.486,A -85,B 0,C 180,E1 -17017.857,E2 -17017.857} C_VEL
LIN {X 0,Y 283.259,Z 315.492,A -85,B 0,C 180,E1 -17020.002,E2 -17020.002} C_VEL
LIN {X 0,Y 284.095,Z 310.358,A -85,B 0,C 180,E1 -17022.138,E2 -17022.138} C_VEL
LIN {X 0,Y 285.053,Z 305.094,A -85,B 0,C 180,E1 -17023.909,E2 -17023.909} C_VEL
LIN {X 0,Y 286.228,Z 298.774,A -85,B 0,C 180,E1 -17025.669,E2 -17025.669} C_VEL
LIN {X 0,Y 287.58,Z 291.723,A -85,B 0,C 180,E1 -17027.301,E2 -17027.301} C_VEL
LIN {X 0,Y 288.794,Z 283.969,A -85,B 0,C 180,E1 -17028.811,E2 -17028.811} C_VEL
LIN {X 0,Y 290.288,Z 275.439,A -85,B 0,C 180,E1 -17030.181,E2 -17030.181} C_VEL
LIN {X 0,Y 291.433,Z 267.843,A -85,B 0,C 180,E1 -17031.206,E2 -17031.206} C_VEL
LIN {X 0,Y 290.906,Z 259.632,A -85,B 0,C 180,E1 -17032.268,E2 -17032.268} C_VEL
LIN {X 0,Y 289.848,Z 250.364,A -85,B 0,C 180,E1 -17033.32,E2 -17033.32} C_VEL
LIN {X 0,Y 288.417,Z 241.537,A -85,B 0,C 180,E1 -17034.198,E2 -17034.198} C_VEL
LIN {X 0,Y 286.03,Z 230.847,A -85,B 0,C 180,E1 -17035.124,E2 -17035.124} C_VEL
LIN {X 0,Y 283.331,Z 221.238,A -85,B 0,C 180,E1 -17035.843,E2 -17035.843} C_VEL
LIN {X 0,Y 283.219,Z 220.222,A -85,B 0,C 180,E1 -17035.914,E2 -17035.914} C_VEL
LIN {X 0,Y 283.751,Z 216.244,A -85,B 0,C 180,E1 -17039.9,E2 -17039.9} C_VEL
LIN {X 0,Y 284.185,Z 213.284,A -85,B 0,C 180,E1 -17042.96,E2 -17042.96} C_VEL
LIN {X 0,Y 284.76,Z 210.152,A -85,B 0,C 180,E1 -17046.322,E2 -17046.322} C_VEL
LIN {X 0,Y 285.378,Z 206.688,A -85,B 0,C 180,E1 -17050.231,E2 -17050.231} C_VEL
LIN {X 0,Y 285.536,Z 203.946,A -85,B 0,C 180,E1 -17053.564,E2 -17053.564} C_VEL
LIN {X 0,Y 285.343,Z 201.806,A -85,B 0,C 180,E1 -17056.397,E2 -17056.397} C_VEL
LIN {X 0,Y 284.952,Z 199.211,A -85,B 0,C 180,E1 -17060.113,E2 -17060.113} C_VEL
LIN {X 0,Y 284.582,Z 196.405,A -85,B 0,C 180,E1 -17064.583,E2 -17064.583} C_VEL
LIN {X 0,Y 284.352,Z 194.932,A -85,B 0,C 180,E1 -17067.175,E2 -17067.175} C_VEL
LIN {X 0,Y 284.354,Z 194.567,A -85,B 0,C 180,E1 -17070.375,E2 -17070.375} C_VEL
LIN {X 0,Y 284.373,Z 194.563,A -85,B 0,C 180,E1 -17073.585,E2 -17073.585} C_VEL
LIN {X 0,Y 284.367,Z 194.567,A -85,B 0,C 180,E1 -17076.706,E2 -17076.706} C_VEL
LIN {X 0,Y 284.4,Z 194.558,A -85,B 0,C 180,E1 -17081.261,E2 -17081.261} C_VEL
LIN {X 0,Y 284.476,Z 194.55,A -85,B 0,C 180,E1 -17084.469,E2 -17084.469} C_VEL
LIN {X 0,Y 284.484,Z 194.548,A -85,B 0,C 180,E1 -17088.601,E2 -17088.601} C_VEL
LIN {X 0,Y 284.636,Z 194.529,A -85,B 0,C 180,E1 -17091.48,E2 -17091.48} C_VEL
LIN {X 0,Y 284.592,Z 194.534,A -85,B 0,C 180,E1 -17094.33,E2 -17094.33} C_VEL
LIN {X 0,Y 284.851,Z 194.499,A -85,B 0,C 180,E1 -17098.585,E2 -17098.585} C_VEL
LIN {X 0,Y 284.851,Z 194.491,A -85,B 0,C 180,E1 -17101.413,E2 -17101.413} C_VEL
LIN {X 0,Y 284.682,Z 194.523,A -85,B 0,C 180,E1 -17107.09,E2 -17107.09} C_VEL
LIN {X 0,Y 284.514,Z 194.541,A -85,B 0,C 180,E1 -17109.956,E2 -17109.956} C_VEL
LIN {X 0,Y 284.477,Z 194.545,A -85,B 0,C 180,E1 -17114.302,E2 -17114.302} C_VEL
LIN {X 0,Y 284.421,Z 194.558,A -85,B 0,C 180,E1 -17117.248,E2 -17117.248} C_VEL
LIN {X 0,Y 284.374,Z 194.556,A -85,B 0,C 180,E1 -17120.242,E2 -17120.242} C_VEL
LIN {X 0,Y 284.364,Z 194.56,A -85,B 0,C 180,E1 -17123.875,E2 -17123.875} C_VEL
LIN {X 0,Y 284.395,Z 194.56,A -85,B 0,C 180,E1 -17127.174,E2 -17127.174} C_VEL
LIN {X 0,Y 284.29,Z 194.571,A -85,B 0,C 180,E1 -17131.274,E2 -17131.274} C_VEL
LIN {X 0,Y 284.356,Z 194.562,A -85,B 0,C 180,E1 -17135.354,E2 -17135.354} C_VEL
LIN {X 0,Y 284.324,Z 194.568,A -85,B 0,C 180,E1 -17138.166,E2 -17138.166} C_VEL
LIN {X 0,Y 284.287,Z 194.572,A -85,B 0,C 180,E1 -17141.872,E2 -17141.872} C_VEL
LIN {X 0,Y 284.251,Z 194.579,A -85,B 0,C 180,E1 -17146.189,E2 -17146.189} C_VEL
LIN {X 0,Y 284.302,Z 194.572,A -85,B 0,C 180,E1 -17150.024,E2 -17150.024} C_VEL
LIN {X 0,Y 284.332,Z 194.567,A -85,B 0,C 180,E1 -17153.615,E2 -17153.615} C_VEL
LIN {X 0,Y 284.305,Z 194.57,A -85,B 0,C 180,E1 -17157.189,E2 -17157.189} C_VEL
LIN {X 0,Y 284.358,Z 194.565,A -85,B 0,C 180,E1 -17160.377,E2 -17160.377} C_VEL
LIN {X 0,Y 284.4,Z 194.615,A -85,B 0,C 180,E1 -17163.89,E2 -17163.89} C_VEL
LIN {X 0,Y 285.408,Z 197.435,A -85,B 0,C 180,E1 -17164.067,E2 -17164.067} C_VEL
LIN {X 0,Y 291.694,Z 210.467,A -85,B 0,C 180,E1 -17165.134,E2 -17165.134} C_VEL
LIN {X 0,Y 296.824,Z 219.164,A -85,B 0,C 180,E1 -17166.075,E2 -17166.075} C_VEL
LIN {X 0,Y 303.044,Z 227.72,A -85,B 0,C 180,E1 -17167.197,E2 -17167.197} C_VEL
LIN {X 0,Y 311.273,Z 237.875,A -85,B 0,C 180,E1 -17168.732,E2 -17168.732} C_VEL
LIN {X 0,Y 319.316,Z 246.89,A -85,B 0,C 180,E1 -17170.389,E2 -17170.389} C_VEL
LIN {X 0,Y 325.464,Z 253.489,A -85,B 0,C 180,E1 -17171.826,E2 -17171.826} C_VEL
LIN {X 0,Y 331.941,Z 260.009,A -85,B 0,C 180,E1 -17173.463,E2 -17173.463} C_VEL
LIN {X 0,Y 337.47,Z 265.434,A -85,B 0,C 180,E1 -17175.059,E2 -17175.059} C_VEL
LIN {X 0,Y 341.385,Z 268.888,A -85,B 0,C 180,E1 -17176.268,E2 -17176.268} C_VEL
LIN {X 0,Y 347.07,Z 274.176,A -85,B 0,C 180,E1 -17178.317,E2 -17178.317} C_VEL
LIN {X 0,Y 350.452,Z 276.687,A -85,B 0,C 180,E1 -17179.602,E2 -17179.602} C_VEL
LIN {X 0,Y 353.007,Z 278.919,A -85,B 0,C 180,E1 -17180.836,E2 -17180.836} C_VEL
LIN {X 0,Y 355.032,Z 280.986,A -85,B 0,C 180,E1 -17182.035,E2 -17182.035} C_VEL
LIN {X 0,Y 356.863,Z 282.6,A -85,B 0,C 180,E1 -17183.214,E2 -17183.214} C_VEL
LIN {X 0,Y 359.667,Z 284.431,A -85,B 0,C 180,E1 -17185.233,E2 -17185.233} C_VEL
LIN {X 0,Y 361.359,Z 285.094,A -85,B 0,C 180,E1 -17186.655,E2 -17186.655} C_VEL
LIN {X 0,Y 362.328,Z 285.419,A -85,B 0,C 180,E1 -17187.777,E2 -17187.777} C_VEL
LIN {X 0,Y 363.01,Z 285.51,A -85,B 0,C 180,E1 -17188.891,E2 -17188.891} C_VEL
LIN {X 0,Y 363.193,Z 285.57,A -85,B 0,C 180,E1 -17190,E2 -17190} C_VEL
LIN {X 0,Y 363.019,Z 285.486,A -85,B 0,C 180,E1 -17191.109,E2 -17191.109} C_VEL
LIN {X 0,Y 362.328,Z 285.401,A -85,B 0,C 180,E1 -17192.223,E2 -17192.223} C_VEL
LIN {X 0,Y 361.356,Z 285.083,A -85,B 0,C 180,E1 -17193.345,E2 -17193.345} C_VEL
LIN {X 0,Y 359.674,Z 284.435,A -85,B 0,C 180,E1 -17194.78,E2 -17194.78} C_VEL
LIN {X 0,Y 356.899,Z 282.56,A -85,B 0,C 180,E1 -17196.785,E2 -17196.785} C_VEL
LIN {X 0,Y 354.903,Z 280.811,A -85,B 0,C 180,E1 -17198.063,E2 -17198.063} C_VEL
LIN {X 0,Y 352.122,Z 278.071,A -85,B 0,C 180,E1 -17199.635,E2 -17199.635} C_VEL
LIN {X 0,Y 348.69,Z 275.506,A -85,B 0,C 180,E1 -17201.042,E2 -17201.042} C_VEL
LIN {X 0,Y 345.308,Z 272.61,A -85,B 0,C 180,E1 -17202.333,E2 -17202.333} C_VEL
LIN {X 0,Y 340.46,Z 268.097,A -85,B 0,C 180,E1 -17204.025,E2 -17204.025} C_VEL
LIN {X 0,Y 335.561,Z 263.44,A -85,B 0,C 180,E1 -17205.547,E2 -17205.547} C_VEL
LIN {X 0,Y 328.506,Z 256.633,A -85,B 0,C 180,E1 -17207.428,E2 -17207.428} C_VEL
LIN {X 0,Y 321.342,Z 249.117,A -85,B 0,C 180,E1 -17209.151,E2 -17209.151} C_VEL
LIN {X 0,Y 315.13,Z 242.251,A -85,B 0,C 180,E1 -17210.501,E2 -17210.501} C_VEL
LIN {X 0,Y 308.851,Z 234.92,A -85,B 0,C 180,E1 -17211.732,E2 -17211.732} C_VEL
LIN {X 0,Y 300.321,Z 224.122,A -85,B 0,C 180,E1 -17213.292,E2 -17213.292} C_VEL
LIN {X 0,Y 294.377,Z 215.26,A -85,B 0,C 180,E1 -17214.371,E2 -17214.371} C_VEL
LIN {X 0,Y 289.806,Z 206.737,A -85,B 0,C 180,E1 -17215.204,E2 -17215.204} C_VEL
LIN {X 0,Y 284.563,Z 195.454,A -85,B 0,C 180,E1 -17216.071,E2 -17216.071} C_VEL
LIN {X 0,Y 284.386,Z 194.563,A -85,B 0,C 180,E1 -17216.135,E2 -17216.135} C_VEL
LIN {X 0,Y 284.314,Z 194.572,A -85,B 0,C 180,E1 -17220.1,E2 -17220.1} C_VEL
LIN {X 0,Y 284.302,Z 194.57,A -85,B 0,C 180,E1 -17222.945,E2 -17222.945} C_VEL
LIN {X 0,Y 284.351,Z 194.565,A -85,B 0,C 180,E1 -17226.383,E2 -17226.383} C_VEL
LIN {X 0,Y 284.347,Z 194.566,A -85,B 0,C 180,E1 -17229.987,E2 -17229.987} C_VEL
LIN {X 0,Y 284.252,Z 194.576,A -85,B 0,C 180,E1 -17234.193,E2 -17234.193} C_VEL
LIN {X 0,Y 284.287,Z 194.572,A -85,B 0,C 180,E1 -17238.128,E2 -17238.128} C_VEL
LIN {X 0,Y 284.324,Z 194.568,A -85,B 0,C 180,E1 -17241.834,E2 -17241.834} C_VEL
LIN {X 0,Y 284.319,Z 194.571,A -85,B 0,C 180,E1 -17245.353,E2 -17245.353} C_VEL
LIN {X 0,Y 284.29,Z 194.571,A -85,B 0,C 180,E1 -17248.726,E2 -17248.726} C_VEL
LIN {X 0,Y 284.395,Z 194.56,A -85,B 0,C 180,E1 -17252.826,E2 -17252.826} C_VEL
LIN {X 0,Y 284.361,Z 194.563,A -85,B 0,C 180,E1 -17256.707,E2 -17256.707} C_VEL
LIN {X 0,Y 284.399,Z 194.559,A -85,B 0,C 180,E1 -17261.262,E2 -17261.262} C_VEL
LIN {X 0,Y 284.488,Z 194.547,A -85,B 0,C 180,E1 -17264.46,E2 -17264.46} C_VEL
LIN {X 0,Y 284.483,Z 194.55,A -85,B 0,C 180,E1 -17268.602,E2 -17268.602} C_VEL
LIN {X 0,Y 284.634,Z 194.527,A -85,B 0,C 180,E1 -17271.481,E2 -17271.481} C_VEL
LIN {X 0,Y 284.593,Z 194.536,A -85,B 0,C 180,E1 -17274.332,E2 -17274.332} C_VEL
LIN {X 0,Y 284.851,Z 194.491,A -85,B 0,C 180,E1 -17278.587,E2 -17278.587} C_VEL
LIN {X 0,Y 284.851,Z 194.499,A -85,B 0,C 180,E1 -17281.415,E2 -17281.415} C_VEL
LIN {X 0,Y 284.683,Z 194.522,A -85,B 0,C 180,E1 -17287.091,E2 -17287.091} C_VEL
LIN {X 0,Y 284.516,Z 194.547,A -85,B 0,C 180,E1 -17289.958,E2 -17289.958} C_VEL
LIN {X 0,Y 284.475,Z 194.55,A -85,B 0,C 180,E1 -17294.304,E2 -17294.304} C_VEL
LIN {X 0,Y 284.423,Z 194.555,A -85,B 0,C 180,E1 -17297.249,E2 -17297.249} C_VEL
LIN {X 0,Y 284.382,Z 194.561,A -85,B 0,C 180,E1 -17300.004,E2 -17300.004} C_VEL
LIN {X 0,Y 283.743,Z 194.647,A -85,B 0,C 180,E1 -17301.187,E2 -17301.187} C_VEL
LIN {X 0,Y 280.866,Z 195.006,A -85,B 0,C 180,E1 -17303.112,E2 -17303.112} C_VEL
LIN {X 0,Y 278.414,Z 195.307,A -85,B 0,C 180,E1 -17304.677,E2 -17304.677} C_VEL
LIN {X 0,Y 277.378,Z 195.434,A -85,B 0,C 180,E1 -17305.89,E2 -17305.89} C_VEL
LIN {X 0,Y 277.305,Z 195.441,A -85,B 0,C 180,E1 -17306.301,E2 -17306.301} C_VEL
LIN {X 0,Y 277.271,Z 195.449,A -85,B 0,C 180,E1 -17310.482,E2 -17310.482} C_VEL
LIN {X 0,Y 277.267,Z 195.71,A -85,B 0,C 180,E1 -17312.162,E2 -17312.162} C_VEL
LIN {X 0,Y 277.599,Z 197.785,A -85,B 0,C 180,E1 -17315.891,E2 -17315.891} C_VEL
LIN {X 0,Y 277.872,Z 199.825,A -85,B 0,C 180,E1 -17319.221,E2 -17319.221} C_VEL
LIN {X 0,Y 278.271,Z 202.373,A -85,B 0,C 180,E1 -17322.994,E2 -17322.994} C_VEL
LIN {X 0,Y 278.42,Z 203.827,A -85,B 0,C 180,E1 -17325.027,E2 -17325.027} C_VEL
LIN {X 0,Y 278.502,Z 205.379,A -85,B 0,C 180,E1 -17327.052,E2 -17327.052} C_VEL
LIN {X 0,Y 278.36,Z 207.119,A -85,B 0,C 180,E1 -17329.24,E2 -17329.24} C_VEL
LIN {X 0,Y 277.849,Z 210.001,A -85,B 0,C 180,E1 -17332.623,E2 -17332.623} C_VEL
LIN {X 0,Y 277.26,Z 213.118,A -85,B 0,C 180,E1 -17336.107,E2 -17336.107} C_VEL
LIN {X 0,Y 276.731,Z 216.491,A -85,B 0,C 180,E1 -17339.711,E2 -17339.711} C_VEL
LIN {X 0,Y 276.221,Z 220.097,A -85,B 0,C 180,E1 -17343.406,E2 -17343.406} C_VEL
LIN {X 0,Y 278.506,Z 228.549,A -85,B 0,C 180,E1 -17344.031,E2 -17344.031} C_VEL
LIN {X 0,Y 280.714,Z 237.591,A -85,B 0,C 180,E1 -17344.811,E2 -17344.811} C_VEL
LIN {X 0,Y 282.597,Z 247.32,A -85,B 0,C 180,E1 -17345.774,E2 -17345.774} C_VEL
LIN {X 0,Y 283.828,Z 257.501,A -85,B 0,C 180,E1 -17346.922,E2 -17346.922} C_VEL
LIN {X 0,Y 284.499,Z 266.493,A -85,B 0,C 180,E1 -17348.093,E2 -17348.093} C_VEL
LIN {X 0,Y 284.463,Z 270.338,A -85,B 0,C 180,E1 -17348.629,E2 -17348.629} C_VEL
LIN {X 0,Y 282.438,Z 281.838,A -85,B 0,C 180,E1 -17350.371,E2 -17350.371} C_VEL
LIN {X 0,Y 280.948,Z 289.936,A -85,B 0,C 180,E1 -17351.914,E2 -17351.914} C_VEL
LIN {X 0,Y 279.623,Z 297.185,A -85,B 0,C 180,E1 -17353.576,E2 -17353.576} C_VEL
LIN {X 0,Y 278.366,Z 303.726,A -85,B 0,C 180,E1 -17355.376,E2 -17355.376} C_VEL
LIN {X 0,Y 277.454,Z 308.228,A -85,B 0,C 180,E1 -17356.822,E2 -17356.822} C_VEL
LIN {X 0,Y 276.517,Z 313.725,A -85,B 0,C 180,E1 -17359.011,E2 -17359.011} C_VEL
LIN {X 0,Y 275.836,Z 318.055,A -85,B 0,C 180,E1 -17361.207,E2 -17361.207} C_VEL
LIN {X 0,Y 275.526,Z 320.424,A -85,B 0,C 180,E1 -17362.673,E2 -17362.673} C_VEL
LIN {X 0,Y 275.352,Z 322.691,A -85,B 0,C 180,E1 -17364.523,E2 -17364.523} C_VEL
LIN {X 0,Y 275.262,Z 324.681,A -85,B 0,C 180,E1 -17367.073,E2 -17367.073} C_VEL
LIN {X 0,Y 275.254,Z 325.272,A -85,B 0,C 180,E1 -17368.537,E2 -17368.537} C_VEL
LIN {X 0,Y 275.254,Z 325.272,A -85,B 0,C 180,E1 -17371.463,E2 -17371.463} C_VEL
LIN {X 0,Y 275.262,Z 324.681,A -85,B 0,C 180,E1 -17372.927,E2 -17372.927} C_VEL
LIN {X 0,Y 275.381,Z 322.228,A -85,B 0,C 180,E1 -17375.859,E2 -17375.859} C_VEL
LIN {X 0,Y 275.685,Z 319.274,A -85,B 0,C 180,E1 -17378.06,E2 -17378.06} C_VEL
LIN {X 0,Y 276.245,Z 315.28,A -85,B 0,C 180,E1 -17380.258,E2 -17380.258} C_VEL
LIN {X 0,Y 277.105,Z 310.146,A -85,B 0,C 180,E1 -17382.449,E2 -17382.449} C_VEL
LIN {X 0,Y 278.147,Z 304.882,A -85,B 0,C 180,E1 -17384.262,E2 -17384.262} C_VEL
LIN {X 0,Y 279.348,Z 298.562,A -85,B 0,C 180,E1 -17386.066,E2 -17386.066} C_VEL
LIN {X 0,Y 280.588,Z 292.611,A -85,B 0,C 180,E1 -17387.492,E2 -17387.492} C_VEL
LIN {X 0,Y 281.715,Z 285.677,A -85,B 0,C 180,E1 -17388.924,E2 -17388.924} C_VEL
LIN {X 0,Y 283.185,Z 277.496,A -85,B 0,C 180,E1 -17390.331,E2 -17390.331} C_VEL
LIN {X 0,Y 284.632,Z 268.984,A -85,B 0,C 180,E1 -17391.548,E2 -17391.548} C_VEL
LIN {X 0,Y 284.122,Z 260.22,A -85,B 0,C 180,E1 -17392.735,E2 -17392.735} C_VEL
LIN {X 0,Y 283.037,Z 250.545,A -85,B 0,C 180,E1 -17393.877,E2 -17393.877} C_VEL
LIN {X 0,Y 281.599,Z 241.959,A -85,B 0,C 180,E1 -17394.774,E2 -17394.774} C_VEL
LIN {X 0,Y 279.172,Z 231.117,A -85,B 0,C 180,E1 -17395.757,E2 -17395.757} C_VEL
LIN {X 0,Y 276.312,Z 220.868,A -85,B 0,C 180,E1 -17396.555,E2 -17396.555} C_VEL
LIN {X 0,Y 276.219,Z 220.002,A -85,B 0,C 180,E1 -17396.644,E2 -17396.644} C_VEL
LIN {X 0,Y 276.754,Z 216.248,A -85,B 0,C 180,E1 -17400.523,E2 -17400.523} C_VEL
LIN {X 0,Y 277.259,Z 213.115,A -85,B 0,C 180,E1 -17403.893,E2 -17403.893} C_VEL
LIN {X 0,Y 277.852,Z 209.967,A -85,B 0,C 180,E1 -17407.376,E2 -17407.376} C_VEL
LIN {X 0,Y 278.371,Z 206.892,A -85,B 0,C 180,E1 -17411.026,E2 -17411.026} C_VEL
LIN {X 0,Y 278.5,Z 205.321,A -85,B 0,C 180,E1 -17412.96,E2 -17412.96} C_VEL
LIN {X 0,Y 278.42,Z 203.77,A -85,B 0,C 180,E1 -17415.025,E2 -17415.025} C_VEL
LIN {X 0,Y 278.028,Z 200.765,A -85,B 0,C 180,E1 -17419.317,E2 -17419.317} C_VEL
LIN {X 0,Y 277.572,Z 197.764,A -85,B 0,C 180,E1 -17424.117,E2 -17424.117} C_VEL
LIN {X 0,Y 277.267,Z 195.71,A -85,B 0,C 180,E1 -17427.838,E2 -17427.838} C_VEL
LIN {X 0,Y 277.266,Z 195.449,A -85,B 0,C 180,E1 -17431.209,E2 -17431.209} C_VEL
LIN {X 0,Y 277.31,Z 195.447,A -85,B 0,C 180,E1 -17434.478,E2 -17434.478} C_VEL
LIN {X 0,Y 277.289,Z 195.447,A -85,B 0,C 180,E1 -17437.654,E2 -17437.654} C_VEL
LIN {X 0,Y 277.343,Z 195.439,A -85,B 0,C 180,E1 -17440.765,E2 -17440.765} C_VEL
LIN {X 0,Y 277.425,Z 195.426,A -85,B 0,C 180,E1 -17445.325,E2 -17445.325} C_VEL
LIN {X 0,Y 277.458,Z 195.425,A -85,B 0,C 180,E1 -17449.786,E2 -17449.786} C_VEL
LIN {X 0,Y 277.637,Z 195.399,A -85,B 0,C 180,E1 -17452.728,E2 -17452.728} C_VEL
LIN {X 0,Y 277.817,Z 195.375,A -85,B 0,C 180,E1 -17458.55,E2 -17458.55} C_VEL
LIN {X 0,Y 277.817,Z 195.366,A -85,B 0,C 180,E1 -17461.449,E2 -17461.449} C_VEL
LIN {X 0,Y 277.636,Z 195.402,A -85,B 0,C 180,E1 -17467.271,E2 -17467.271} C_VEL
LIN {X 0,Y 277.457,Z 195.419,A -85,B 0,C 180,E1 -17470.212,E2 -17470.212} C_VEL
LIN {X 0,Y 277.43,Z 195.424,A -85,B 0,C 180,E1 -17474.674,E2 -17474.674} C_VEL
LIN {X 0,Y 277.34,Z 195.436,A -85,B 0,C 180,E1 -17479.233,E2 -17479.233} C_VEL
LIN {X 0,Y 277.315,Z 195.438,A -85,B 0,C 180,E1 -17484.17,E2 -17484.17} C_VEL
LIN {X 0,Y 277.323,Z 195.439,A -85,B 0,C 180,E1 -17487.506,E2 -17487.506} C_VEL
LIN {X 0,Y 277.267,Z 195.448,A -85,B 0,C 180,E1 -17490.481,E2 -17490.481} C_VEL
LIN {X 0,Y 277.249,Z 195.447,A -85,B 0,C 180,E1 -17493.894,E2 -17493.894} C_VEL
LIN {X 0,Y 277.28,Z 195.444,A -85,B 0,C 180,E1 -17497.466,E2 -17497.466} C_VEL
LIN {X 0,Y 277.229,Z 195.451,A -85,B 0,C 180,E1 -17501.232,E2 -17501.232} C_VEL
LIN {X 0,Y 277.199,Z 195.454,A -85,B 0,C 180,E1 -17505.226,E2 -17505.226} C_VEL
LIN {X 0,Y 277.218,Z 195.452,A -85,B 0,C 180,E1 -17509.512,E2 -17509.512} C_VEL
LIN {X 0,Y 277.269,Z 195.447,A -85,B 0,C 180,E1 -17512.532,E2 -17512.532} C_VEL
LIN {X 0,Y 277.243,Z 195.452,A -85,B 0,C 180,E1 -17516.104,E2 -17516.104} C_VEL
LIN {X 0,Y 277.257,Z 195.45,A -85,B 0,C 180,E1 -17519.539,E2 -17519.539} C_VEL
LIN {X 0,Y 277.336,Z 195.439,A -85,B 0,C 180,E1 -17523.188,E2 -17523.188} C_VEL
LIN {X 0,Y 278.434,Z 198.445,A -85,B 0,C 180,E1 -17523.389,E2 -17523.389} C_VEL
LIN {X 0,Y 284.8,Z 212.013,A -85,B 0,C 180,E1 -17524.556,E2 -17524.556} C_VEL
LIN {X 0,Y 289.243,Z 220.171,A -85,B 0,C 180,E1 -17525.457,E2 -17525.457} C_VEL
LIN {X 0,Y 295.827,Z 229.977,A -85,B 0,C 180,E1 -17526.778,E2 -17526.778} C_VEL
LIN {X 0,Y 304.025,Z 240.234,A -85,B 0,C 180,E1 -17528.41,E2 -17528.41} C_VEL
LIN {X 0,Y 312.215,Z 249.706,A -85,B 0,C 180,E1 -17530.1,E2 -17530.1} C_VEL
LIN {X 0,Y 319.575,Z 257.556,A -85,B 0,C 180,E1 -17531.783,E2 -17531.783} C_VEL
LIN {X 0,Y 325.592,Z 263.727,A -85,B 0,C 180,E1 -17533.297,E2 -17533.297} C_VEL
LIN {X 0,Y 331.443,Z 269.37,A -85,B 0,C 180,E1 -17534.945,E2 -17534.945} C_VEL
LIN {X 0,Y 337.109,Z 274.527,A -85,B 0,C 180,E1 -17536.743,E2 -17536.743} C_VEL
LIN {X 0,Y 340.896,Z 278.061,A -85,B 0,C 180,E1 -17538.103,E2 -17538.103} C_VEL
LIN {X 0,Y 344.331,Z 280.782,A -85,B 0,C 180,E1 -17539.415,E2 -17539.415} C_VEL
LIN {X 0,Y 347.153,Z 283.04,A -85,B 0,C 180,E1 -17540.68,E2 -17540.68} C_VEL
LIN {X 0,Y 349.26,Z 285.171,A -85,B 0,C 180,E1 -17541.903,E2 -17541.903} C_VEL
LIN {X 0,Y 351.148,Z 286.895,A -85,B 0,C 180,E1 -17543.103,E2 -17543.103} C_VEL
LIN {X 0,Y 353.065,Z 288.289,A -85,B 0,C 180,E1 -17544.426,E2 -17544.426} C_VEL
LIN {X 0,Y 354.43,Z 289.074,A -85,B 0,C 180,E1 -17545.451,E2 -17545.451} C_VEL
LIN {X 0,Y 355.805,Z 289.624,A -85,B 0,C 180,E1 -17546.603,E2 -17546.603} C_VEL
LIN {X 0,Y 356.824,Z 289.949,A -85,B 0,C 180,E1 -17547.742,E2 -17547.742} C_VEL
LIN {X 0,Y 357.536,Z 290.045,A -85,B 0,C 180,E1 -17548.874,E2 -17548.874} C_VEL
LIN {X 0,Y 357.744,Z 290.093,A -85,B 0,C 180,E1 -17550,E2 -17550} C_VEL
LIN {X 0,Y 357.538,Z 290.028,A -85,B 0,C 180,E1 -17551.126,E2 -17551.126} C_VEL
LIN {X 0,Y 356.823,Z 289.932,A -85,B 0,C 180,E1 -17552.258,E2 -17552.258} C_VEL
LIN {X 0,Y 355.804,Z 289.613,A -85,B 0,C 180,E1 -17553.397,E2 -17553.397} C_VEL
LIN {X 0,Y 354.449,Z 289.069,A -85,B 0,C 180,E1 -17554.549,E2 -17554.549} C_VEL
